Omron CX-Programmer project NuevoProyecto (CX-Programmer 9.80)

# PLC NuevoPLC1: CJ2M CPU34
I/O table (CPU CJ2M-CPU34): rack 0 slot 0 CJ1W-ID211; rack 0 slot 1 CJ1W-ID211; rack 0 slot 2 CJ1W-ID211; rack 0 slot 3 CJ1W-ID211; rack 0 slot 4 CJ1W-OD212; rack 0 slot 5 CJ1W-OD212; rack 0 slot 6 CJ1W-OC211; rack 0 slot 7 CJ1W-CT021; rack 0 slot 11 CJ2M-EIP21

## Global symbols (name address type ; comment)
Alta_vel_Motor_carro_film 6.04 BOOL  ; Alta velocidad del motor de arrastre
Aplicador_desplazado 0.03 BOOL  ; DT. Aplicador desplazado
Aplicador_en_reposo 0.02 BOOL  ; DT. Aplicador en reposo
0.11 BOOL  ; Llave en campo habilita cinta inclinana
0.12 BOOL  ; Run Variador V1 (falla=0)
0.13 BOOL  ; Run variador V2 (falla=0)
0.14 BOOL  ; run variador V3 (falla=0)
0.15 BOOL  ; Señal monitor de tensión (falla=0)
1000.00 BOOL  ; Manual/Automático
1001.00 BOOL  ; Paradas General
108.00 BOOL  ; Entrada de bolsa
10.00 BOOL  ; Ciclo Rodillos - Paso 0 - muevo rodillos
11.00 BOOL  ; Ciclo rodillos - Muevo rodillos hasta centrador
120.00 BOOL  ; Activación de Resto
121.00 BOOL  ; Secuencia resto - Paso 1
122.00 BOOL  ; Secuencia resto - Paso 2
123.00 BOOL  ; Secuencia resto - Paso 3
124.00 BOOL  ; Secuencia resto - Paso 4
125.00 BOOL  ; Secuencia resto  - Paso 5
126.00 BOOL  ; Secuencia resto - Paso 6
128.00 BOOL  ; Se hizo resto
129.00 BOOL  ; Señal fin transferencia enfundadora
12.00 BOOL  ; Ciclo rodillos - Paso 2 -muevo rodillos
135.00 BOOL  ; Deshabilitado
138.00 BOOL  ; Carro pala fin avanse
139.00 BOOL  ; Carro pala - segundo avance
13.00 BOOL  ; Ciclo rodillos - paso 3 - mover Rodillos
144.00 BOOL  ; Primer avance carro pala
145.00 BOOL  ; Segundo avance carro pala
146.00 BOOL  ; Primer avance carro pala
147.00 BOOL  ; segundo avance carro pala
14.00 BOOL  ; Ciclo rodillos - Paso 4 - entrada pallet elevador mover rodillos cuando elevador abajop
150.00 BOOL  ; Sensor
150.01 BOOL  ; Activar bandera
150.05 BOOL  ; Auxiliar Sensor
155.00 BOOL  ; Fin extracto
156.00 BOOL  ; Fin extracto
15.00 BOOL  ; Ciclo rodillos - Paso 5 - Habilita subir pallet, muevo rodillo
16.00 BOOL  ; Ciclo rodillos - paso 6 - muevo rodillos salida pallets
17.00 BOOL  ; Secuencia rodillos - Ultimo paso (necesita puas abajo)
18.00 BOOL  ; Pallet subio en elevador
2000.00 BOOL  ; Alarma por falta de run V1
2000.01 BOOL  ; alarma por falla de run V2
2000.02 BOOL  ; Alarma por falta de run V3
2000.03 BOOL  ; Alarma por falla en alimentación
2000.04 BOOL  ; Alarma por falla de guardamotor D1
2000.05 BOOL  ; Alarma por falla de guardamotor D2
2000.06 BOOL  ; Alarma por falla de gaurdamotor D5
2000.07 BOOL  ; Alarma por falla de guardamotor D7
2000.08 BOOL  ; Alarma por falla variador Elevador
2000.09 BOOL  ; Alarma por falla guardamotor D8L
2000.10 BOOL  ; Alarma por falla guardamotor D9
2000.15 BOOL  ; Falla en motores (termicos)
2001.00 BOOL  ; Flash en HMI
2001.01 BOOL  ; Falla en motores (termicos)
2002.00 BOOL  ; P_emergencia 1 pulsado
2002.01 BOOL  ; P_emergencia 2 pulsado
2002.02 BOOL  ; P_emergencia 3 pulsado
2002.03 BOOL  ; P_emergencia 4 pulsado
2002.04 BOOL  ; Swicht seguridad 1
2002.05 BOOL  ; Swicht seguridad 2
2002.06 BOOL  ; Swicht seguridad 3
2002.07 BOOL  ; Swicht seguridad 4
2002.08 BOOL  ; Swicht seguridad 5
2002.09 BOOL  ; Cortina de seguridad
2002.10 BOOL  ; Contactor alimentación general caido
2002.11 BOOL  ; Discrepancia en entrada de PLC seguridad
2002.12 BOOL  ; Discrepancia en salida de PLC seguridad
2002.13 BOOL  ; Maquina sin seguridad
2002.14 BOOL  ; Barrera inhibida
2002.15 BOOL  ; Pulsador de emregencia pallet vacios pulsada
2003.00 BOOL  ; flash HMI
2004.00 BOOL  ; Pulsador de emergencia escalera
2004.01 BOOL  ; Barrera de seguridad entrada de Pallets
2004.02 BOOL  ; Seguridad de Barrera entrada de Pallets Inhibida
200.00 BOOL  ; Elevador bajar rapido
200.01 BOOL  ; Elevador subir rapido
200.02 BOOL  ; Elevador bajar lento
200.03 BOOL  ; Elevador subir lento
200.05 BOOL  ; Elevador subir rapido
200.06 BOOL  ; Elevador subir rapido
200.07 BOOL  ; Auxiliar freno
2010.00 BOOL  ; Flash en HMI
202.00 BOOL  ; Deformación
2100.00 BOOL  ; Open Gate counter 1
2101.01 BOOL  ; Close gate counter 1
2102.00 BOOL  ; gate open
2102.01 BOOL  ; Gate Close
2102.03 BOOL  ; Reset counter 1
2122 CHANNEL  ; Counter1 (módulo CT021)
250.00 BOOL  ; Habilito  tarea Automatico
250.01 BOOL  ; Habilito tarea Manual
250.02 BOOL  ; Habilito tarea seguridad
29.00 BOOL  ; Auxiliar ciclo elevador - ok para meter pallet
300.00 BOOL  ; Marcha Automático
301.00 BOOL  ; Automático activo
302.00 BOOL  ; M MANUAL
30.00 BOOL  ; Ciclo elevador - paso 0 - bajar lento
31.00 BOOL  ; Ciclo elevador - Paso 1 - Subir rapido
32.00 BOOL  ; Ciclo elevador - Paso 2 - subir rapido
33.00 BOOL  ; Ciclo elevador - subir lento
34.00 BOOL  ; Ciclo elevador - Paso 4 - Bajar lento
35.00 BOOL  ; Ciclo elevador - Paso 5 - Subir lento
36.00 BOOL  ; Ciclo elevador - paso 6 - bajar lento
37.00 BOOL  ; Ciclo elevador - Paso 7 - bajar..lento...rapido
38.00 BOOL  ; Ciclo elevador - Paso 8 - Bajar rapido lento, Fin pallets
39.00 BOOL  ; Cambio de pallets
3.07 BOOL  ; Señal guardamotor D1 (falla=0)
3.08 BOOL  ; Señal guardamotor D2 (falla=0)
3.09 BOOL  ; Señal guardamotor D5 (falla=0)
3.10 BOOL  ; Señal guardamotor D7 (falla=0)
3.11 BOOL  ; Señal guardamotor C8R (falla=0)
3.12 BOOL  ; Señal guardamotor D8L (falla=0)
3.13 BOOL  ; Señal guardamotor D9 (falla=0)
3.15 BOOL  ; FT vacia
400.00 BOOL  ; Función puesta a cero
400.01 BOOL  ; Paso 1 - carro hacia atrás
400.02 BOOL  ; Paso 2 - caro hacia delante libera sensor
400.03 BOOL  ; Paso 3 - Tiempo
400.04 BOOL  ; Paso 4 - Retrocede carro hasta sensor
400.05 BOOL  ; Paso 5 -  reset encoder
400.06 BOOL  ; Paso 6 - Tiempo para poner 0
400.10 BOOL  ; Cero carro OK
401.00 BOOL  ; Baja velocidad carro
401.01 BOOL  ; Velocidad alta de carro
402.00 BOOL  ; Sujeta FIlm (=1 sujetando)
403.00 BOOL  ; Pinzas (=1 cierra)
404.00 BOOL  ; Corte lamina
404.01 BOOL  ; Retorno de cuchilla
405.00 BOOL  ; Auxiliar sensor pallet
405.01 BOOL  ; Auxiliar
408.00 BOOL  ; Film colocado
40.00 BOOL  ; Inicio ciclo pallet
41.00 BOOL  ; Al medio y salir
42.00 BOOL  ; Ya afuera subir
43.00 BOOL  ; Alimentación de pallet
44.00 BOOL  ; Ir abajo y entrar
45.00 BOOL  ; Sensor en medio
46.00 BOOL  ; bolsa colgada
500.00 BOOL  ; Ya salió pallet
501.00 BOOL  ; Terminó secuencia resto
50.00 BOOL  ; Comando cerrar compuerta
51.00 BOOL  ; Comando abrir compuerta
52.00 BOOL  ; Compuerta abierta
54.00 BOOL  ; Bandera para realizar bolsa 4,8,12 y 16
55.00 BOOL  ; Bolsa 4, 8, 12 y 16 en posicion
57.00 BOOL  ; Palet en elevador
58.00 BOOL  ; Activación de barrera
599.14 BOOL  ; P_Off
5.08 BOOL  ; Bandela elevador
600.00 BOOL  ; Activación manual HMI
600.01 BOOL  ; Desactivación Manual HMI
600.02 BOOL  ; Llave Man Aut HMI (1=AUT)
600.04 BOOL  ; Marcha Automático HMI
600.05 BOOL  ; Puesta a cero HMI
600.06 BOOL  ; Resto
600.07 BOOL  ; Cambio de pallets
600.10 BOOL  ; Boton reset HMI
60.00 BOOL  ; Paso 0 - Carro pala Esperando bolsas
610.00 BOOL  ; Manual HMI alimentador
610.01 BOOL  ; Manual HMI Calefactores/ventilalor
610.02 BOOL  ; Manual avance HMI
610.03 BOOL  ; Manual retroceso HMI
610.04 BOOL  ; Manual HMI Prensa
610.05 BOOL  ; Manual pinza HMI
610.06 BOOL  ; Manual corte HMI
610.07 BOOL  ; Manual HMI centrador derecho
610.08 BOOL  ; Manual centrador izquierdo HMI
610.10 BOOL  ; Boton reconocimiento HMI
61.00 BOOL  ; Paso 1 - carro pala avance
62.00 BOOL  ; Paso 2  - carro pala avanza un poco mas (presiona bolsa)
63.00 BOOL  ; paso 3 - Carro pala retroceder
64.00 BOOL  ; Auxiliar sacar banderas de pedido
65.00 BOOL  ; Bandera de realizar avance de carro pala
68.00 BOOL  ; Pulsos de carro pala > Activación de velocidad carro pala
69.00 BOOL  ; Se realizo secuencia avance Bolsa 8 y 16
6.01 BOOL  ; Motor transporte rodillos film
6.14 BOOL  ; Cilindros sujeta Film en elevador
6.15 BOOL  ; Reserva cableada
700.00 BOOL  ; Fin Avance de carro pala (en pulsos)
70.00 BOOL  ; Primera secuencia hecha
72.00 BOOL  ; Seguridad arrastre carro pala
76.00 BOOL  ; Bolsa entrando (filtros con sensores)
77.00 BOOL  ; Pulso para decodificador de movimiento rodillos (bolsas)
800.00 BOOL  ; Auxiliar
82.00 BOOL  ; Pulso bolsa par entrando
86.00 BOOL  ; Rodillos superiores movio OK
87.00 BOOL  ; Bolsas impares
88.00 BOOL  ; Bolsas pares
90.00 BOOL  ; Solicitud de accionamiento de tope de giro
91.00 BOOL  ; Accionar tope de giro (demora encendido)
92.00 BOOL  ; Accionar tope de giro (demora apagado)
93.00 BOOL  ; Solicitud de accionar valvula desplazadora
94.00 BOOL  ; Accionar desplazador
950.00 BOOL  ; M Manual/automático
95.00 BOOL  ; M dosificación
C0014 BOOL  ; C dosificador
D100 CHANNEL  ; Pasos secuencia Maquina Film
D1000 CHANNEL  ; HMI - CANTIDAD DE FILAS POR PALLET
D1002 CHANNEL  ; Filas de pallets
D1003 CHANNEL  ; Activación de velocidad carro pala
D1005 CHANNEL  ; Cantidad pulsos de Avance de carro
D101 CHANNEL  ; Paso anterior
D1012 CHANNEL  ; Pisos en donde se activa la secuencia de carga de pallet
D1014 CHANNEL  ; Pulsos a realizar cinta programada
D200 CHANNEL  ; Programa seleccionado en HMI
D2000 CHANNEL  ; Encoder en milimetros
D2002 CHANNEL  ; Destino en mm de carro
D2004 CHANNEL  ; Largo HMI
D2006 CHANNEL  ; Segundo avance HMI
D2008 CHANNEL  ; Maximo distancia film
D202 CHANNEL  ; Pasos de la secuencia EF
D210 CHANNEL  ; Tiempo desde HMI
D211 CHANNEL  ; Tiempo desde HMI
D212 CHANNEL  ; Tiempo desde HMI
D213 CHANNEL  ; Tiempo desde HMI
D214 CHANNEL  ; Tiempo para seguir arrastre
D300 CHANNEL  ; Decodificador secuencia cargador de pallets
D3100.00 BOOL  ; Comunicacion PLC seg. Inhibir barrera
D3100.01 BOOL  ; Comunicacion PLC seg. Inhibir barrera entrada de Pallets
D3100.02 BOOL  ; Señal para G9SP - Aviso Hay movimmientos
D3100.03 BOOL  ; Señal para G9SP - Espero Inicio de Ciclo de Pallets se habiliat a cargar
D400 CHANNEL  ; Decodificador secuencia rodillos
D406 CHANNEL  ; Tiempo HMI
D410 CHANNEL  ; Decodificador secuencia rodillos salida
D420 CHANNEL  ; Decodificador salida
D500 CHANNEL  ; Bolsa 1
D5000 CHANNEL  ; Contador bolsas
D5002 CHANNEL  ; Bolsas
D5004 CHANNEL  ; Auxiliar
D5006 CHANNEL  ; Rodillos de pallets
D5008 CHANNEL  ; Cantidad de pisos realizados
D501 CHANNEL  ; Bolsa 2
D5010 CHANNEL  ; Cantidad de pisos realizados
D5012 CHANNEL  ; Auxiliar
D5014 CHANNEL  ; Auxiliar
D5016 CHANNEL  ; Auxiliar
D5018 CHANNEL  ; Auxiliar contador 6
D502 CHANNEL  ; Bolsa 3
D5020 CHANNEL  ; Pulsos carro pala
D5022 CHANNEL  ; Auxiliar c7
D5024 CHANNEL  ; Auxiliar c8 (Accionamiento rodillos superiores)
D5026 CHANNEL  ; Pulsos tope de giro
D5028 CHANNEL  ; Auxiliar C11
D503 CHANNEL  ; Bolsa 4
D5030 CHANNEL  ; Demora de accion de desplazador
D5032 CHANNEL  ; Contador cinta programada
D505 CHANNEL  ; Bolsa 6
D507 CHANNEL  ; Bolsa 8
D508 CHANNEL  ; Bolsa 9
D509 CHANNEL  ; Bolsa 10
D510 CHANNEL  ; Bolsa 11
D5100 CHANNEL  ; Contador
D5102 CHANNEL  ; Contador salida
D512 CHANNEL  ; Bolsa 13
D513 CHANNEL  ; Bolsa 14
D514 CHANNEL  ; Bolsa 15
D6000 CHANNEL  ; Pulsos/tiempo para parar rodillos
H0.01 BOOL  ; Pallet Euro=1  Pallet standar=0(HMI)
H0.05 BOOL  ; Enfundadora NO habilitada - HMI
H0.15 BOOL  ; PUENTE 3.15
H10.00 BOOL  ; Habilitacion de Euro Pallet
T0001 BOOL  ; Tiempo, señal habilita salida pallets
T0002 BOOL  ; Elevador abajo
T0003 BOOL  ; Demora de Nivelacion
T0004 BOOL  ; Tiempo de bolsa colgada
T0005 BOOL  ; Tiempo libera fotocelula nivelacion
T0006 BOOL  ; Demora de dosificacion
T0007 BOOL  ; T. compuerta cerrada
T0009 BOOL  ; Tiempo compuerta abierta
T0010 BOOL  ; Tiempo espera pala arriba (filtro)
T0011 BOOL  ; Tiempo carros
T0020 BOOL  ; Tiempo Automático
T0022 BOOL  ; Tiempo centrada
T0030 BOOL  ; Auxiliar freno
T0031 BOOL  ; Auxiliar liberó freno
T0050 BOOL  ; Demora rodillos superior
T0100 BOOL  ; Tiempo apagado ventilador, seguridad calefactores
T0101 BOOL  ; Tiempo centrado longitudinal pallet
T0102 BOOL  ; Tiempo centrado Euro pallet
T0103 BOOL  ; Tiempo espera accionar centrado
T0104 BOOL  ; Tiempo centrado
T0105 BOOL  ; Tiempo centrado
T0106 BOOL  ; Tiempo espera cierre pinzas
T0107 BOOL  ; Espera apertura
T0108 BOOL  ; Tiempo espera corte
T0109 BOOL  ; Tiempo espera avance
T0110 BOOL  ; Tiempo pequeño avance
T0111 BOOL  ; Tiempo espera avance final
T0112 BOOL  ; Tiempo avance sin film
T0113 BOOL  ; Espera retroceso
T0114 BOOL  ; tiempo de calentado film
T0115 BOOL  ; Tiempo calentado film
T0116 BOOL  ; Tiempo falla, pallet trabado
T0120 BOOL  ; Filtro acumulacion de pallets
T0200 BOOL  ; Tiempo auxiliar
T0201 BOOL  ; Tiempo auxiliar
T0202 BOOL  ; Auxiliar
T0203 BOOL  ; Auxiliar
T0204 BOOL  ; Auxiliar
T0205 BOOL  ; Tiempo falla
T0206 BOOL  ; Auxiliar
T0207 BOOL  ; Auxiliar
T0208 BOOL  ; Auxiliar
T0209 BOOL  ; Auxiliar
T0210 BOOL  ; Auxiliar
T0211 BOOL  ; T auxiliar alarma
T0212 BOOL  ; Auxiliar
T0213 BOOL  ; Auxiliar
T0214 BOOL  ; Tiempo para alarma
T0215 BOOL  ; Tiempo para hacer 0
T0216 BOOL  ; T auxiliar alarma
T0217 BOOL  ; Auxiliar
T0218 BOOL  ; Auxiliar
T0219 BOOL  ; Auxiliar
T0220 BOOL  ; Auxiliar
T0221 BOOL  ; Auxiliar
T0222 BOOL  ; Auxiliar
T0223 BOOL  ; Auxiliar
T0224 BOOL  ; Auxiliar no hay pallet
T0225 BOOL  ; Auxiliar
T0226 BOOL  ; Auxiliar
T0227 BOOL  ; Centrador longitudinal
T0228 BOOL  ; Auxiliar tiempo centrador activo
T0229 BOOL  ; Auxiliar
T0230 BOOL  ; auxiliar
T0231 BOOL  ; Auxiliar
T0232 BOOL  ; auxiliar
T0233 BOOL  ; Auxiliar liberacion
T0234 BOOL  ; Auxiliar falla
T0235 BOOL  ; Auxiliar
T0236 BOOL  ; T espera liberación
T0237 BOOL  ; Auxiliar filtro ensor
T0238 BOOL  ; Auxiliar
T0239 BOOL  ; T subir bandela
T0240 BOOL  ; Auxiliar
T0242 BOOL  ; Auxiliar
T0243 BOOL  ; Auxiliar
T0244 BOOL  ; T auxiliar
T1016 BOOL  ; Tiempo de secado de pallets
W12 CHANNEL  ; Salida decodicicador EF
W121.00 BOOL  ; Salida decodificador 3
W121.01 BOOL  ; Salida decodificador 3
W121.02 BOOL  ; Salida decodificador 3
W121.03 BOOL  ; Salida decodificador 3
W121.04 BOOL  ; Salida decodificador 3
W121.05 BOOL  ; Salida decodificador 3
W121.06 BOOL  ; Salida decodificador 3
W121.07 BOOL  ; Salida decodificador 3
W121.08 BOOL  ; Salida decodificador 3
W121.09 BOOL  ; Salida decodificador 3
W121.10 BOOL  ; Salida decodificador 3
W121.11 BOOL  ; Salida decodificador 3
W121.12 BOOL  ; Salida decodificador 3
W121.13 BOOL  ; Salida decodificador 3
W121.14 BOOL  ; Salida decodificador 3
W121.15 BOOL  ; Salida decodificador 3
W150.00 BOOL  ; Paso  0 - Inicio
W150.02 BOOL  ; Paso 2 - Espero OK cinta anterior
W150.04 BOOL  ; Muevo hasta sensor
W150.05 BOOL  ; Paso 5 - Movimiento OK de Cinta
W150.06 BOOL  ; Paso 6 - movimiento OK - Secuencia entrada elevador
W150.08 BOOL  ; Paso 8 - entrar a elevador
W150.10 BOOL  ; Paso 10 - Tiempo
W150.12 BOOL  ; Paso 12 - Pallet dentro de elevador
W150.14 BOOL  ; Paso 14 - movimiento salida
W151.00 BOOL  ; Paso 16 - entrando nuevo pallet
W151.02 BOOL  ; Paso 18 - Pallet ok para elevador
W151.04 BOOL  ; Paso 20 . Salida de pallet
W151.06 BOOL  ; Paso 22 - salida pallets
W151.09 BOOL  ; paso 25 - Alarma pallet trabado
W151.10 BOOL  ; Paso 26 - Alarma de pallet trabado
W200 CHANNEL  ; Canal secuencia maq film
W201 CHANNEL  ; Canal secuencia maq film
W202.00 BOOL  ; Encender cinta rodillos film
W202.01 BOOL  ; Centar pallet derecho Euro
W202.02 BOOL  ; Centar pallet izquierdo Euro
W202.03 BOOL  ; Centar pallet derecho STD
W202.04 BOOL  ; Centar pallets izquierdo STD
W202.05 BOOL  ; Retraer cilindro centrador derecho
W202.06 BOOL  ; Retraer cilindro centrador izquierdo
W202.07 BOOL  ; Val. prensa (mordaza)
W202.08 BOOL  ; Valvula pinzas
W202.09 BOOL  ; Arrastre avance
W202.10 BOOL  ; Motor alimentación film
W202.11 BOOL  ; Corte hacia la izquierda=1 corte hacia la derecha=0
W202.12 BOOL  ; Pequeño avance
W202.13 BOOL  ; Avance sin film (corto)
W202.14 BOOL  ; Arrastre Retroceso
W202.15 BOOL  ; Auxiliar precalentar (paso 2)
W203.00 BOOL  ; Encender rodillos film con rodillos
W203.01 BOOL  ; Habilito secuencia nuevo pallets (habilito finalización de secuencia pallets)
W203.02 BOOL  ; Auxiliar cortar hacia la derecha
W203.03 BOOL  ; Cortador hacia la izquierda
W204.00 BOOL  ; Motor ventilador
W204.01 BOOL  ; Calefactores
W250.01 BOOL  ; Paso 1 - espero
W250.02 BOOL  ; paso 2 -
W250.03 BOOL  ; Paso 3 - Espero reposición enfundadora
W250.04 BOOL  ; paso 4
W250.05 BOOL  ; Paso 5 - Espero OK enfundadora
W300.00 BOOL  ; Paso 0 maquina Film
W300.01 BOOL  ; Paso 1 - Puesta a cero
W300.02 BOOL  ; Paso 2 - Espera de pallets
W300.03 BOOL  ; Paso 3 - movimiento de rodillos
W300.04 BOOL  ; Paso 4 - Centrador de pallets
W300.05 BOOL  ; Paso 5 - Tiempo
W300.06 BOOL  ; Paso 6 - Cierre de pinzas
W300.07 BOOL  ; Paso 7 - Tiempo
W300.08 BOOL  ; Paso 8 - Abre sujeta film
W300.09 BOOL  ; Paso 9 - Primer avance de carro
W300.10 BOOL  ; Paso 10 - Cierre sujetador
W300.11 BOOL  ; Paso 11 - corte de lamina
W300.12 BOOL  ; Paso 12 - Segundo avance
W300.13 BOOL  ; Paso 13 - Abrir pinzas
W300.14 BOOL  ; Paso 14 - termino maq film, cero
W300.15 BOOL  ; Paso 15 - Traslado de pallets
W301.00 BOOL  ; Paso 16
W301.01 BOOL  ; Paso 17
W301.02 BOOL  ; Paso 18
W301.03 BOOL  ; Paso 19
W301.04 BOOL  ; Paso 20
W301.05 BOOL  ; Paso 21
W301.06 BOOL  ; Paso 22
W301.07 BOOL  ; Paso 23
W301.08 BOOL  ; Paso 24
W301.09 BOOL  ; Paso 25
W301.10 BOOL  ; Paso 26
W301.11 BOOL  ; Paso 27
W301.12 BOOL  ; Paso 28
W301.13 BOOL  ; Paso 29
W301.14 BOOL  ; Paso 30
W301.15 BOOL  ; Paso 31
W50.00 BOOL  ; Paso 0 - espero Inicio
W50.01 BOOL  ; Paso 1 -entrar puas
W50.02 BOOL  ; Paso 2 - Bajar puas
W50.03 BOOL  ; Paso 3 - Subir puas medio
W50.04 BOOL  ; Paso 4 - Puas salir
W50.05 BOOL  ; Paso 5 - puas subir
W50.06 BOOL  ; Paso 6 - Pallet listo para sacar - Secuencia cargador
W50.07 BOOL  ; Paso 7 - bajar puas
W50.08 BOOL  ; Paso  8 - Entrar puas
W50.09 BOOL  ; Paso  9 - espero reinicio de ciclo
W50.12 BOOL  ; Pallet trabado
W66.01 BOOL  ; CMD MANUAL - SALIR PRENSA LATERAL
W66.02 BOOL  ; STOP PRENSA LATERAL
W80.00 BOOL  ; Paso  0 - espero inicio
W80.02 BOOL  ; Paso 2 - espero Ok cargador para mover
W80.04 BOOL  ; Paso 4 - muevo cintas
W80.06 BOOL  ; Paso 6 - Ok salio pallet de cargado, Muevo cinta film
W80.08 BOOL  ; Paso 8 - activo centrador
W80.10 BOOL  ; Paso 10 - Espero OK de maq film
W80.12 BOOL  ; Paso 12 - pallet listo para sacar
W80.14 BOOL  ; Paso 14 - Falla, pallet trabajo
W90.00 BOOL  ; Paso  0 - Inicio
W90.02 BOOL  ; Paso 2 - Espero OK cinta anterior
W90.04 BOOL  ; Muevo hasta sensor
W90.06 BOOL  ; Paso 6 - movimiento OK
W90.08 BOOL  ; Paso 8 - entrar a elevador
W90.10 BOOL  ; Paso 10 - Tiempo
W90.12 BOOL  ; Paso 12 - Pallet dentro de elevador
W90.14 BOOL  ; Paso 14 - movimiento salida
Contador_1 Conversion_Encoder
Corte_Activo 0.10 BOOL  ; DT. corte aplicador activado
Corte_en_reposo 0.09 BOOL  ; DT. Cortador en reposo
Estado_entradas_G9SP D3007 CHANNEL  ; Estado entradas PLC seguridad (0=falla bit a bit)
Estado_entradas_G9SP_16_19 D3008 CHANNEL  ; Estado entradas PLC seguridad (0=falla bit a bit)
Estado_salidas_G9SP D3010 CHANNEL  ; Estado salidas PLC seguridad (0=falla bit a bit)
Falla_variador_transportador 3.02 BOOL  ; FC PRENSA LATERAL, POS 1
Fallo_variador_arrastre 3.05 BOOL  ; Falla en variador de arrastre de film
Fi_transferenci_enfundadora 0.08 BOOL  ; Fin de trasferencia de pallets a la enfundadora (señal desde enfundadora)
Hab_FILM H0.00 BOOL  ; Habilitación proceso máquina film
I_G9SP_0 D3002.00 BOOL  ; .
I_G9SP_1 D3002.01 BOOL  ; Entrada PLC Seguridad P_emergencia embolsadora payper
I_G9SP_10 D3002.10 BOOL  ; Entrada PLC Seguridad Cortina seguridad 1
I_G9SP_11 D3002.11 BOOL  ; Entrada PLC Seguridad Cortina seguridad 1
I_G9SP_12 D3002.12 BOOL  ; Entrada PLC Seguridad Contacto modo
I_G9SP_13 D3002.13 BOOL  ; Entrada PLC Seguridad Contacto modo
I_G9SP_14 D3002.14 BOOL  ; Entrada PLC Seguridad Realimentacion relé
I_G9SP_15 D3002.15 BOOL  ; Entrada PLC Seguridad
I_G9SP_16 D3003.00 BOOL  ; Entrada PLC Seguridad
I_G9SP_17 D3003.01 BOOL  ; Entrada PLC Seguridad
I_G9SP_18 D3003.02 BOOL  ; Entrada PLC Seguridad
I_G9SP_19 D3003.03 BOOL  ; Entrada PLC Seguridad
I_G9SP_2 D3002.02 BOOL  ; Entrada PLC Seguridad P_emergencia 2 pallet lleno
I_G9SP_3 D3002.03 BOOL  ; Entrada PLC Seguridad P_emergencia 3 estrichadora
I_G9SP_4 D3002.04 BOOL  ; Entrada PLC Seguridad P_emergencia gabinete comando
I_G9SP_5 D3002.05 BOOL  ; Entrada PLC Seguridad Swicht 1 pallet vacio
I_G9SP_6 D3002.06 BOOL  ; Entrada PLC Seguridad Swicht 2 puerta de elevador
I_G9SP_7 D3002.07 BOOL  ; Entrada PLC Seguridad Swicht 3 pallet lleno
I_G9SP_8 D3002.08 BOOL  ; Entrada PLC Seguridad Swicht 4 puerta tablero neumatico
I_G9SP_9 D3002.09 BOOL  ; Entrada PLC Seguridad Swicht 5 puerta tablero comando
Llave_cinta_inclinada 0.11 BOOL  ; Llave cinta inclinada
M976 W121.00 BOOL  ; Salida decodificador 3
M977 W121.01 BOOL  ; Salida decodificador 3
M978 W121.02 BOOL  ; Salida decodificador 3
M979 W121.03 BOOL  ; Salida decodificador 3
M980 W121.04 BOOL  ; Salida decodificador 3
M981 W121.05 BOOL  ; Salida decodificador 3
M982 W121.06 BOOL  ; Salida decodificador 3
M983 W121.07 BOOL  ; Salida decodificador 3
M984 W121.08 BOOL  ; Salida decodificador 3
M985 W121.09 BOOL  ; Salida decodificador 3
M986 W121.10 BOOL  ; Salida decodificador 3
M987 W121.11 BOOL  ; Salida decodificador 3
M988 W121.12 BOOL  ; Salida decodificador 3
M989 W121.13 BOOL  ; Salida decodificador 3
M990 W121.14 BOOL  ; Salida decodificador 3
M991 W121.15 BOOL  ; Salida decodificador 3
Motor_Rodillos_pallets_vacios 5.13 BOOL  ; Motor transporte de rodillos pallets vacios
Motor_alim_film 6.02 BOOL  ; Motor alimentación de film
Motor_avance 6.05 BOOL  ; Motor de arrastre avance (variador)
Motor_retroceso 6.06 BOOL  ; Motor de arrastre retroceso (variador)
Motor_rodillos_film 6.01 BOOL  ; Motor transporte rodillos film
OLD_M160 160.00 BOOL  ; Programa 1
OLD_M161 160.01 BOOL  ; Programa 2
OLD_M960 W120.00 BOOL  ; Salida decodificador 3
OLD_M961 W120.01 BOOL  ; Salida decodificador 3
OLD_M962 W120.02 BOOL  ; Salida decodificador 3
OLD_M963 W120.03 BOOL  ; Salida decodificador 3
OLD_M964 W120.04 BOOL  ; Salida decodificador 3
OLD_M965 W120.05 BOOL  ; Salida decodificador 3
OLD_M966 W120.06 BOOL  ; Salida decodificador 3
OLD_M967 W120.07 BOOL  ; Salida decodificador 3
OLD_M968 W120.08 BOOL  ; Salida decodificador 3
OLD_M969 W120.09 BOOL  ; Salida decodificador 3
OLD_M970 W120.10 BOOL  ; Salida decodificador 3
OLD_M971 W120.11 BOOL  ; Salida decodificador 3
OLD_M972 W120.12 BOOL  ; Salida decodificador 3
OLD_M973 W120.13 BOOL  ; Salida decodificador 3
OLD_M974 W120.14 BOOL  ; Salida decodificador 3
OLD_M975 W120.15 BOOL  ; Salida decodificador 3
OLD_S0 W0.00 BOOL  ; Salida decodificador
OLD_S1 W0.01 BOOL  ; Salida decodificador - Bolsa 1
OLD_S10 W0.10 BOOL  ; Salida decodificador - Bolsa 10
OLD_S100 W100.00 BOOL  ; Salida decodificador 2
OLD_S101 W100.01 BOOL  ; Salida decodificador 2 Entrada de bolsa
OLD_S102 W100.02 BOOL  ; Salida decodificador 2
OLD_S103 W100.03 BOOL  ; Salida decodificador 2
OLD_S104 W100.04 BOOL  ; Salida decodificador 2
OLD_S105 W100.05 BOOL  ; Salida decodificador 2
OLD_S106 W100.06 BOOL  ; Salida decodificador 2
OLD_S107 W100.07 BOOL  ; Salida decodificador 2
OLD_S108 W100.08 BOOL  ; Salida decodificador 2
OLD_S109 W100.09 BOOL  ; Salida decodificador 2
OLD_S11 W0.11 BOOL  ; Salida decodificador - Bolsa 11
OLD_S110 W100.10 BOOL  ; Salida decodificador 2
OLD_S111 W100.11 BOOL  ; Salida decodificador 2
OLD_S112 W100.12 BOOL  ; Salida decodificador 2
OLD_S113 W100.13 BOOL  ; Salida decodificador 2
OLD_S114 W100.14 BOOL  ; Salida decodificador 2
OLD_S115 W100.15 BOOL  ; Salida decodificador 2
OLD_S116 W101.00 BOOL  ; Salida decodificador 2
OLD_S12 W0.12 BOOL  ; Salida decodificador - Bolsa 12
OLD_S13 W0.13 BOOL  ; Salida decodificador - Bolsa 13
OLD_S14 W0.14 BOOL  ; Salida decodificador - Bolsa 14
OLD_S15 W0.15 BOOL  ; Salida decodificador - Bolsa 15
OLD_S16 W1.00 BOOL  ; Salida decodificador - Bolsa 16
OLD_S2 W0.02 BOOL  ; Salida decodificador - Bolsa 2
OLD_S3 W0.03 BOOL  ; Salida decodificador
OLD_S4 W0.04 BOOL  ; Salida decodificador - Bolsa 4
OLD_S5 W0.05 BOOL  ; Salida decodificador - Bolsa 5
OLD_S6 W0.06 BOOL  ; Salida decodificador - Bolsa 6
OLD_S7 W0.07 BOOL  ; Salida decodificador - Bolsa 7
OLD_S8 W0.08 BOOL  ; Salida decodificador - Bolsa 8
OLD_S9 W0.09 BOOL  ; Salida decodificador - Bolsa 9
OLD_X0 1.00 BOOL  ; Control contaje carro pala
OLD_X16 3.03 BOOL  ; PLC seguridad OK=1
OLD_X27 1.02 BOOL  ; FT acumulación sacos
OLD_X30 1.03 BOOL  ; FT dosificación
OLD_X31 1.04 BOOL  ; FT contaje
OLD_X32 1.05 BOOL  ; FT carros
OLD_X33 1.06 BOOL  ; Pala arriba
OLD_X34 1.07 BOOL  ; Carro pala en reposo
OLD_X35 1.08 BOOL  ; Carro Pala sobre compuerta
OLD_X36 1.09 BOOL  ; Carro pala desplazado
OLD_X37 1.10 BOOL  ; Seguridad arraste carro pala
OLD_X4 1.01 BOOL  ; Seg contrapeso
OLD_X40 1.11 BOOL  ; Compuerta abierta
OLD_X41 1.12 BOOL  ; Compuerta cerrada
OLD_X42 1.13 BOOL  ; Deformación compuerta
OLD_X43 1.14 BOOL  ; Elevador arriba
OLD_X44 1.15 BOOL  ; Elevador cambio velocidad subiendo
OLD_X45 2.00 BOOL  ; Elevador cambio velocidad bajando
OLD_X46 2.01 BOOL  ; elevador abajo
OLD_X47 2.02 BOOL  ; Fotocelula nivelación
OLD_X50 2.03 BOOL  ; Puas dentro
OLD_X51 2.04 BOOL  ; Puas fuera
OLD_X52 2.05 BOOL  ; Puas arriba
OLD_X53 2.06 BOOL  ; Puas centro
OLD_X54 2.07 BOOL  ; Puas abajo
OLD_X55 2.08 BOOL  ; FT. Pallet en espera
OLD_X56 2.09 BOOL  ; FT seguridad entrada elevador
OLD_X57 2.10 BOOL  ; FT pallet en elevador
OLD_X60 2.11 BOOL  ; FT seguridad salida elevador
OLD_X61 2.12 BOOL  ; Acumulación pallets lleno
OLD_X63 2.14 BOOL  ; Presion aire
OLD_X64 2.15 BOOL  ; Valvula desplazadora afuera
OLD_X65 3.00 BOOL  ; Valvula desplazadora adentro
OLD_X66 3.06 BOOL  ; Señal de OK de enfundadora no listo
OLD_Y0 4.00 BOOL  ; Cinta inclinada
OLD_Y1 4.01 BOOL  ; Cinta aplanado superior (Paralaelo inferior)
OLD_Y10 4.08 BOOL  ; Carro pala velocidad 1
OLD_Y11 4.09 BOOL  ; Carro pala velocidad 2
OLD_Y12 4.10 BOOL  ; EV. SALE PRENSA LATERAL
OLD_Y13 4.11 BOOL  ; Desplazador Cinta programada-Alinear. (Válvula)
OLD_Y14 4.12 BOOL  ; Abrir compuerta
OLD_Y15 4.13 BOOL  ; Cerrar compuerta
OLD_Y16 5.00 BOOL  ; Multivelocidad variador (velocidad rápida)
OLD_Y17 5.01 BOOL  ; Freno de elevador
OLD_Y2 4.02 BOOL  ; Cinta Programada
OLD_Y20 4.14 BOOL  ; Elevador subir
OLD_Y21 4.15 BOOL  ; Elevador bajar
OLD_Y22 5.02 BOOL  ; Rodillos palets
OLD_Y23 5.03 BOOL  ; Puas entrar (válvula)
OLD_Y24 5.04 BOOL  ; Puas salir (válvula)
OLD_Y25 5.05 BOOL  ; Puas bajar (válvulas)
OLD_Y26 5.06 BOOL  ; Puas Subir (válvula)
OLD_Y27 5.07 BOOL  ; Barrera (válvula)
OLD_Y3 4.03 BOOL  ; Tope de giro (válvula)
OLD_Y30 6.10 BOOL  ; Centrado pallets (válvula)
OLD_Y31 5.09 BOOL  ; Señal paletizadora en marcha
OLD_Y32 5.10 BOOL  ; Baliza verde
OLD_Y33 5.11 BOOL  ; Baliza Rojo
OLD_Y34 5.12 BOOL  ; EV. ENTRA PRENSA LATERAL
OLD_Y35 6.01 BOOL  ; Salida libre
OLD_Y36 5.14 BOOL  ; Señal para enfundadora - No enfundar
OLD_Y37 5.15 BOOL  ; señal para máquina estrichadora
OLD_Y4 4.04 BOOL  ; Rodillos Superiores
OLD_Y5 4.05 BOOL  ; Pala (válvula)
OLD_Y6 4.06 BOOL  ; Avanzar carro pala
OLD_Y7 4.07 BOOL  ; Retroceder carro pala
O_G9SP_0 D3005.00 BOOL  ; Salida PLC Seguridad Piloto P_emergencia 1
O_G9SP_1 D3005.01 BOOL  ; Salida PLC Seguridad Piloto P_emergencia 2
O_G9SP_2 D3005.02 BOOL  ; Salida PLC Seguridad Piloto P_emergencia 3
O_G9SP_3 D3005.03 BOOL  ; Salida PLC Seguridad Piloto P_emergencia 4
O_G9SP_4 D3005.04 BOOL  ; Salida PLC Seguridad Contactor
O_G9SP_5 D3005.05 BOOL  ; Salida PLC Seguridad
O_G9SP_6 D3005.06 BOOL  ; Salida PLC Seguridad
O_G9SP_7 D3005.07 BOOL  ; Salida PLC Seguridad
P0_film W200.00 BOOL  ; Paso 0 (poner maq en reposo)
P10_film W200.10 BOOL
P11_film W200.11 BOOL
P12_film W200.12 BOOL
P13_film W200.13 BOOL
P14_film W200.14 BOOL
P15_film W200.15 BOOL
P1_film W200.01 BOOL  ; Paso 1 (espera de pallets)
P2_film W200.02 BOOL  ; Centrar pallet transversalmente
P3_film W200.03 BOOL  ; Cierra pinzas y abre mordazas
P4_film W200.04 BOOL  ; Arrastre
P5_film W200.05 BOOL  ; Corte
P6_film W200.06 BOOL  ; pequeño avance
P7_film W200.07 BOOL  ; Retroceso y centrado con calor
P8_film W200.08 BOOL  ; Sacado de pallet a cinta siguiente
P9_film W200.09 BOOL
Pallet_en_cargador 2.13 BOOL  ; Pallet en cargador
Permiso_enfundadora 0.07 BOOL  ; Permiso entrar pallets en enfundadadora
Pres_pallet 0.00 BOOL  ; Presencia de pallet en trasnporte (fotocelda)
Pulsador_abrir_sujetador 0.04 BOOL  ; Llave de habilitación
Pulsador_cerrar_sujetador 0.05 BOOL  ; Pulsador Abrir/Cerrar sujetador de Film
Pulsador_parada_cintas 0.06 BOOL  ; Pulsador parada de cintas
Sensor_control_bobina 0.01 BOOL  ; DT. control bobina aplicador
Termico_arrastre_film 3.04 BOOL  ; Termico de arrastre de film
Termico_trasportador 3.01 BOOL  ; Termico transportador aplicador de film
Val_abrir_pinzas 6.08 BOOL  ; Valvulas abrir pinzas aplicador
Val_abrir_sujetador 6.07 BOOL  ; Valvula abrir sujetador de film
Val_corte 6.09 BOOL  ; Valvula corte lamina aplicador
Valvula_centrador 6.10 BOOL  ; Válvula centrado de pallets vaios
Valvula_centrador_der_no 6.11 BOOL  ; Val. Biestable centrador derecho no accionado
Valvula_cerrar_pinzas 6.13 BOOL  ; Valvula cerrar pinzas aplicador
Valvula_cerrar_sujetador 6.12 BOOL  ; Válvula cerrar sujeta Film aplicador
Velocidad_variador Funcion_baja_velocidad
Ventilador_conveccion 6.03 BOOL  ; Ventilador de aire de convección

## Program General (cyclic task 0)
Local symbols
OLD_M976 BOOL
OLD_X015 BOOL
OLD_X140 BOOL
OLD_X142 BOOL

### Section _Inicio_Salto

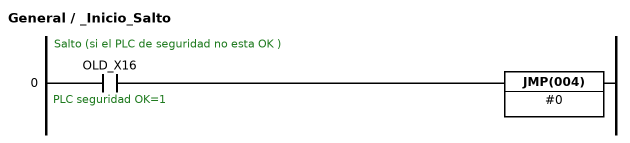
; rung 0: Salto (si el PLC de seguridad no esta OK )
LD OLD_X16  ; PLC seguridad OK=1
JMP(004) #0

### Section Cargador_pallets

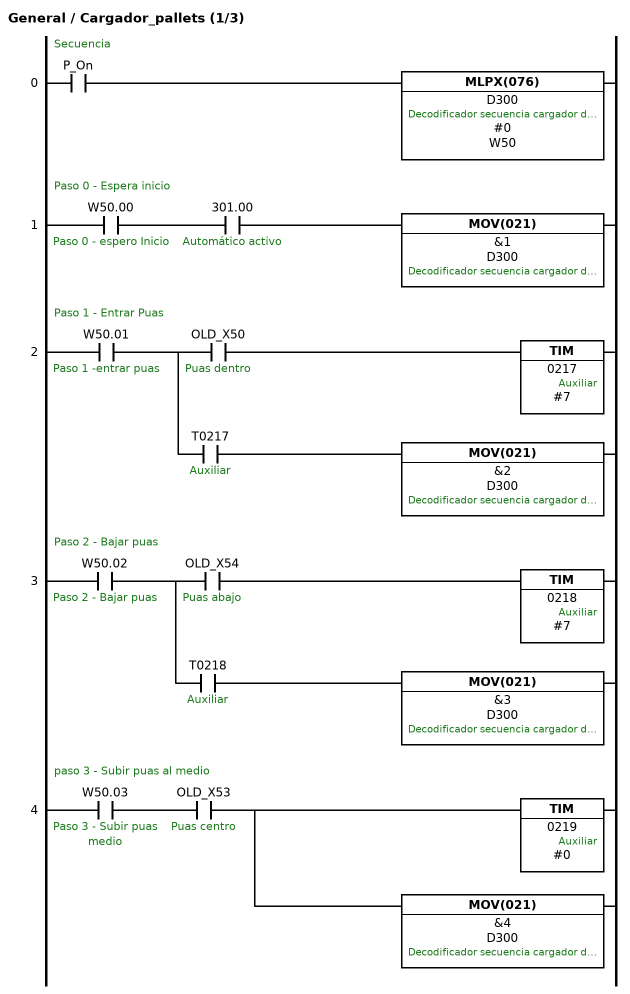
; rung 0: Secuencia
LD P_On
MLPX(076) D300 #0 W50  ; Decodificador secuencia cargador de pallets
; rung 1: Paso 0 - Espera inicio
LD W50.00  ; Paso 0 - espero Inicio
AND 301.00  ; Automático activo
MOV(021) &1 D300  ; Decodificador secuencia cargador de pallets
; rung 2: Paso 1 - Entrar Puas
LD W50.01  ; Paso 1 -entrar puas
OUT TR0
AND OLD_X50  ; Puas dentro
TIM 0217 #7  ; Auxiliar
LD TR0
AND T0217  ; Auxiliar
MOV(021) &2 D300  ; Decodificador secuencia cargador de pallets
; rung 3: Paso 2 - Bajar puas
LD W50.02  ; Paso 2 - Bajar puas
OUT TR0
AND OLD_X54  ; Puas abajo
TIM 0218 #7  ; Auxiliar
LD TR0
AND T0218  ; Auxiliar
MOV(021) &3 D300  ; Decodificador secuencia cargador de pallets
; rung 4: paso 3 - Subir puas al medio
LD W50.03  ; Paso 3 - Subir puas medio
AND OLD_X53  ; Puas centro
TIM 0219 #0  ; Auxiliar
MOV(021) &4 D300  ; Decodificador secuencia cargador de pallets

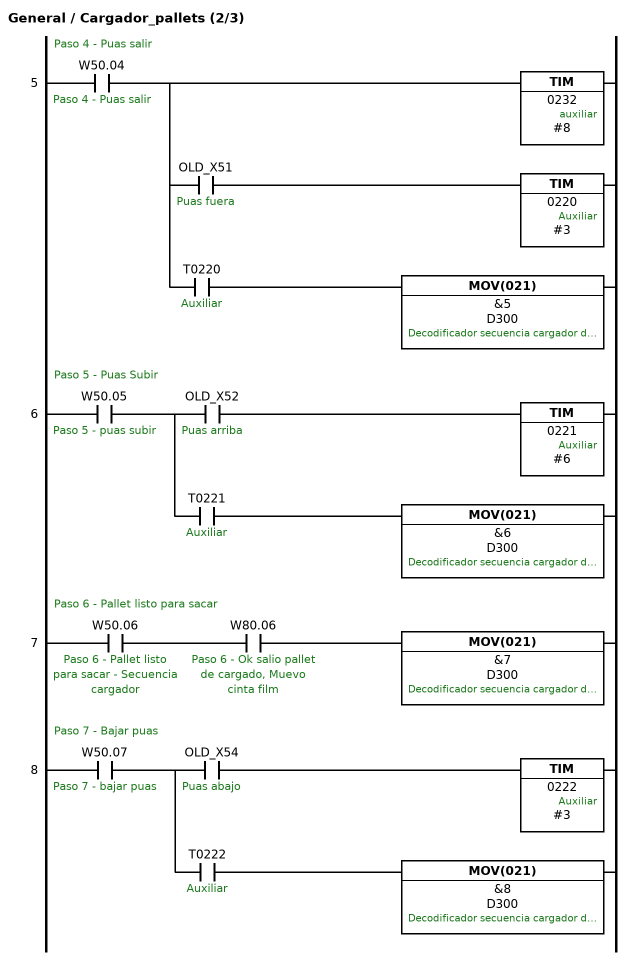
; rung 5: Paso 4 - Puas salir
LD W50.04  ; Paso 4 - Puas salir
OUT TR0
TIM 0232 #8  ; auxiliar
AND OLD_X51  ; Puas fuera
TIM 0220 #3  ; Auxiliar
LD TR0
AND T0220  ; Auxiliar
MOV(021) &5 D300  ; Decodificador secuencia cargador de pallets
; rung 6: Paso 5 - Puas Subir
LD W50.05  ; Paso 5 - puas subir
OUT TR0
AND OLD_X52  ; Puas arriba
TIM 0221 #6  ; Auxiliar
LD TR0
AND T0221  ; Auxiliar
MOV(021) &6 D300  ; Decodificador secuencia cargador de pallets
; rung 7: Paso 6 - Pallet listo para sacar
LD W50.06  ; Paso 6 - Pallet listo para sacar - Secuencia cargador
AND W80.06  ; Paso 6 - Ok salio pallet de cargado, Muevo cinta film
MOV(021) &7 D300  ; Decodificador secuencia cargador de pallets
; rung 8: Paso 7 - Bajar puas
LD W50.07  ; Paso 7 - bajar puas
OUT TR0
AND OLD_X54  ; Puas abajo
TIM 0222 #3  ; Auxiliar
LD TR0
AND T0222  ; Auxiliar
MOV(021) &8 D300  ; Decodificador secuencia cargador de pallets

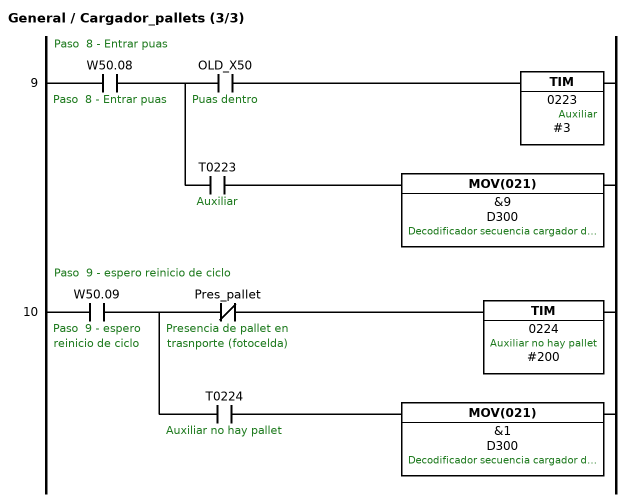
; rung 9: Paso  8 - Entrar puas
LD W50.08  ; Paso  8 - Entrar puas
OUT TR0
AND OLD_X50  ; Puas dentro
TIM 0223 #3  ; Auxiliar
LD TR0
AND T0223  ; Auxiliar
MOV(021) &9 D300  ; Decodificador secuencia cargador de pallets
; rung 10: Paso  9 - espero reinicio de ciclo
LD W50.09  ; Paso  9 - espero reinicio de ciclo
OUT TR0
ANDNOT Pres_pallet  ; Presencia de pallet en trasnporte (fotocelda)
TIM 0224 #200  ; Auxiliar no hay pallet
LD TR0
AND T0224  ; Auxiliar no hay pallet
MOV(021) &1 D300  ; Decodificador secuencia cargador de pallets

### Section Rodillos_centrador

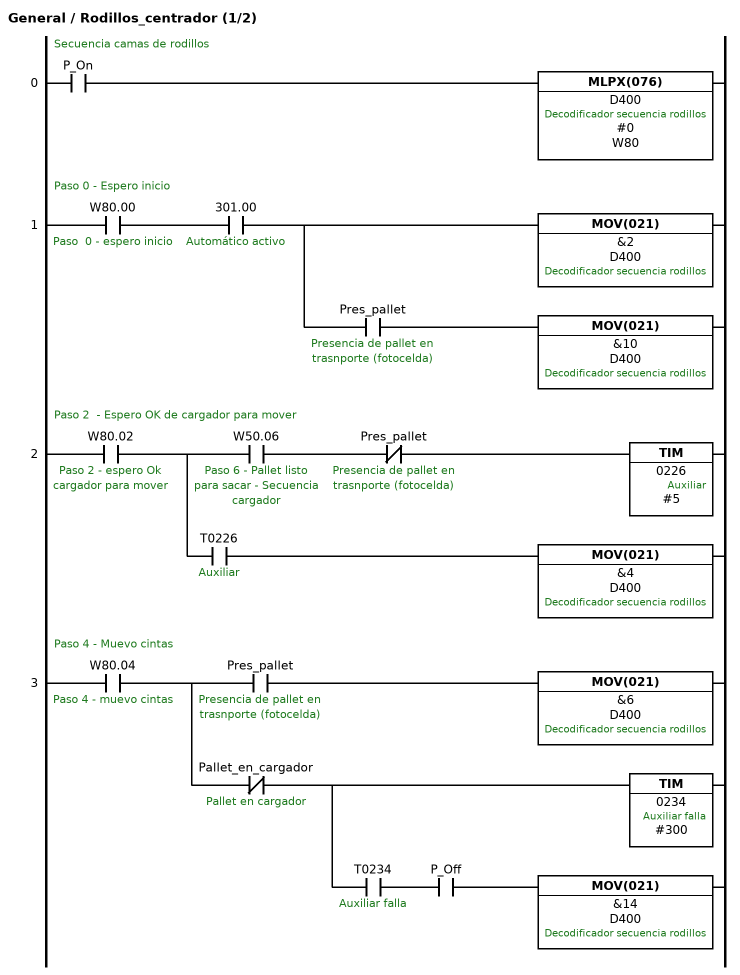
; rung 0: Secuencia camas de rodillos
LD P_On
MLPX(076) D400 #0 W80  ; Decodificador secuencia rodillos
; rung 1: Paso 0 - Espero inicio
LD W80.00  ; Paso  0 - espero inicio
AND 301.00  ; Automático activo
MOV(021) &2 D400  ; Decodificador secuencia rodillos
AND Pres_pallet  ; Presencia de pallet en trasnporte (fotocelda)
MOV(021) &10 D400  ; Decodificador secuencia rodillos
; rung 2: Paso 2  - Espero OK de cargador para mover
LD W80.02  ; Paso 2 - espero Ok cargador para mover
OUT TR0
AND W50.06  ; Paso 6 - Pallet listo para sacar - Secuencia cargador
ANDNOT Pres_pallet  ; Presencia de pallet en trasnporte (fotocelda)
TIM 0226 #5  ; Auxiliar
LD TR0
AND T0226  ; Auxiliar
MOV(021) &4 D400  ; Decodificador secuencia rodillos
; rung 3: Paso 4 - Muevo cintas
LD W80.04  ; Paso 4 - muevo cintas
OUT TR0
AND Pres_pallet  ; Presencia de pallet en trasnporte (fotocelda)
MOV(021) &6 D400  ; Decodificador secuencia rodillos
LD TR0
ANDNOT Pallet_en_cargador  ; Pallet en cargador
TIM 0234 #300  ; Auxiliar falla
AND T0234  ; Auxiliar falla
AND P_Off
MOV(021) &14 D400  ; Decodificador secuencia rodillos

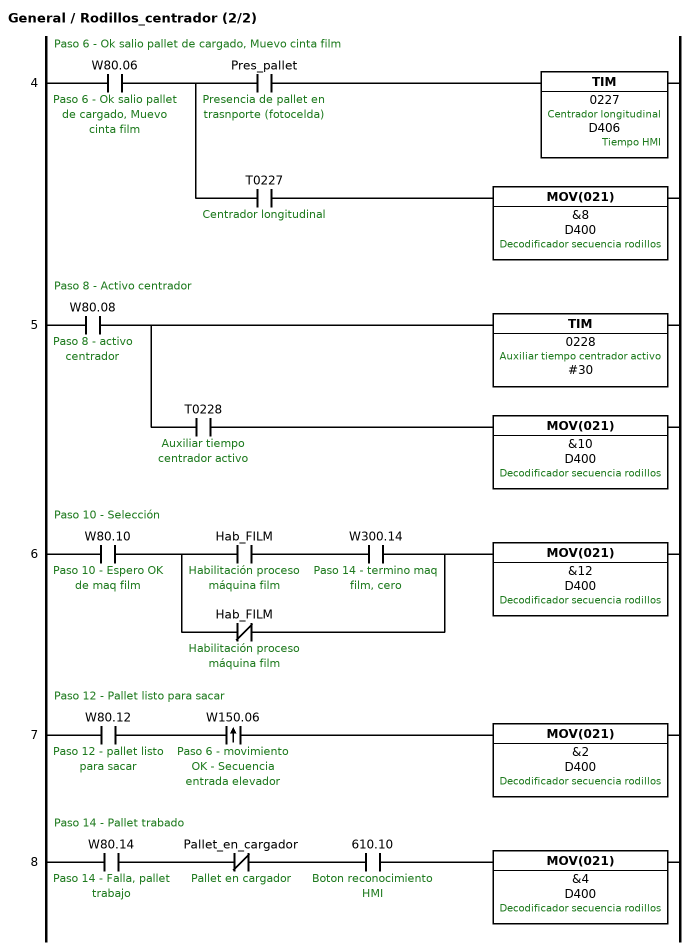
; rung 4: Paso 6 - Ok salio pallet de cargado, Muevo cinta film
LD W80.06  ; Paso 6 - Ok salio pallet de cargado, Muevo cinta film
OUT TR0
AND Pres_pallet  ; Presencia de pallet en trasnporte (fotocelda)
TIM 0227 D406  ; Tiempo HMI, Centrador longitudinal
LD TR0
AND T0227  ; Centrador longitudinal
MOV(021) &8 D400  ; Decodificador secuencia rodillos
; rung 5: Paso 8 - Activo centrador
LD W80.08  ; Paso 8 - activo centrador
TIM 0228 #30  ; Auxiliar tiempo centrador activo
AND T0228  ; Auxiliar tiempo centrador activo
MOV(021) &10 D400  ; Decodificador secuencia rodillos
; rung 6: Paso 10 - Selección
LD W80.10  ; Paso 10 - Espero OK de maq film
LD Hab_FILM  ; Habilitación proceso máquina film
AND W300.14  ; Paso 14 - termino maq film, cero
ORNOT Hab_FILM  ; Habilitación proceso máquina film
ANDLD
MOV(021) &12 D400  ; Decodificador secuencia rodillos
; rung 7: Paso 12 - Pallet listo para sacar
LD W80.12  ; Paso 12 - pallet listo para sacar
@AND W150.06  ; Paso 6 - movimiento OK - Secuencia entrada elevador
MOV(021) &2 D400  ; Decodificador secuencia rodillos
; rung 8: Paso 14 - Pallet trabado
LD W80.14  ; Paso 14 - Falla, pallet trabajo
ANDNOT Pallet_en_cargador  ; Pallet en cargador
AND 610.10  ; Boton reconocimiento HMI
MOV(021) &4 D400  ; Decodificador secuencia rodillos

### Section Rodillos_entrada_elevador

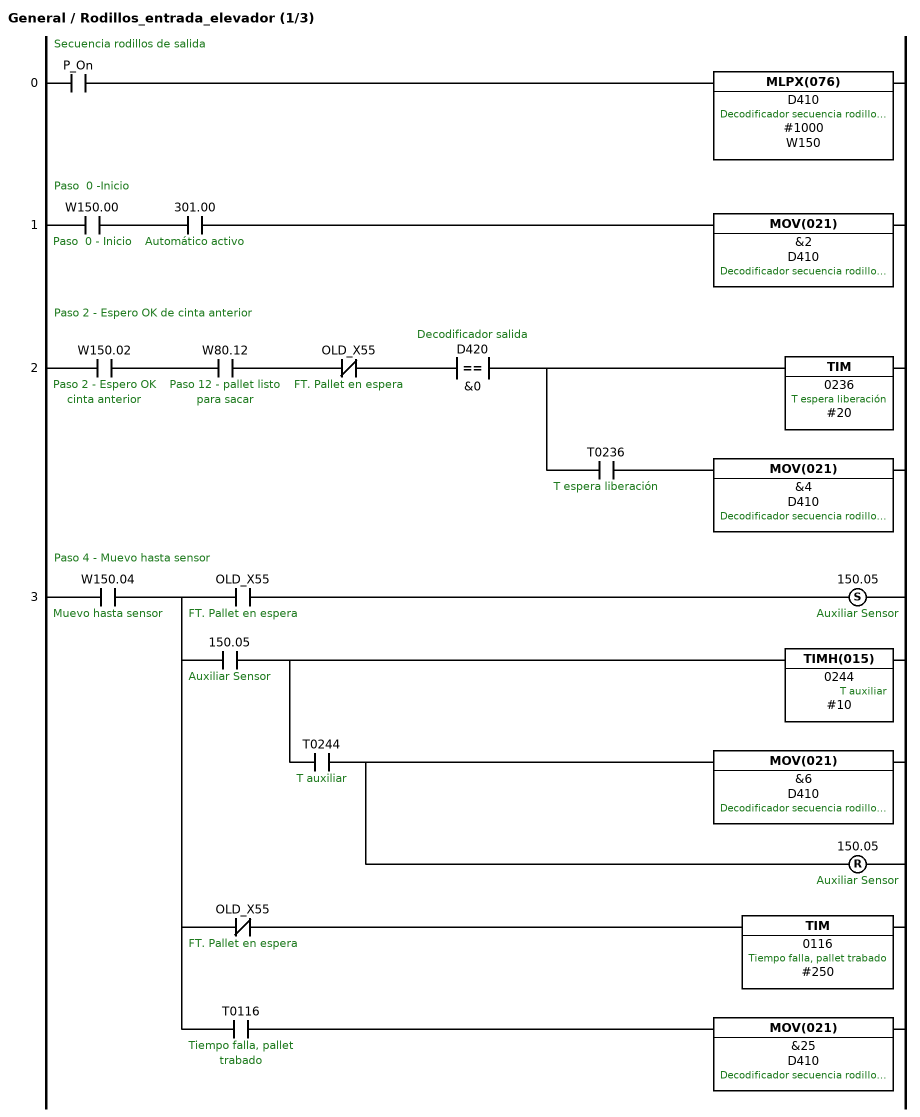
; rung 0: Secuencia rodillos de salida
LD P_On
MLPX(076) D410 #1000 W150  ; Decodificador secuencia rodillos salida
; rung 1: Paso  0 -Inicio
LD W150.00  ; Paso  0 - Inicio
AND 301.00  ; Automático activo
MOV(021) &2 D410  ; Decodificador secuencia rodillos salida
; rung 2: Paso 2 - Espero OK de cinta anterior
LD W150.02  ; Paso 2 - Espero OK cinta anterior
AND W80.12  ; Paso 12 - pallet listo para sacar
ANDNOT OLD_X55  ; FT. Pallet en espera
AND=(300) D420 &0  ; Decodificador salida
TIM 0236 #20  ; T espera liberación
AND T0236  ; T espera liberación
MOV(021) &4 D410  ; Decodificador secuencia rodillos salida
; rung 3: Paso 4 - Muevo hasta sensor
LD W150.04  ; Muevo hasta sensor
OUT TR0
AND OLD_X55  ; FT. Pallet en espera
SET 150.05  ; Auxiliar Sensor
LD TR0
AND 150.05  ; Auxiliar Sensor
TIMH(015) 0244 #10  ; T auxiliar
AND T0244  ; T auxiliar
MOV(021) &6 D410  ; Decodificador secuencia rodillos salida
RSET 150.05  ; Auxiliar Sensor
LD TR0
ANDNOT OLD_X55  ; FT. Pallet en espera
TIM 0116 #250  ; Tiempo falla, pallet trabado
LD TR0
AND T0116  ; Tiempo falla, pallet trabado
MOV(021) &25 D410  ; Decodificador secuencia rodillos salida

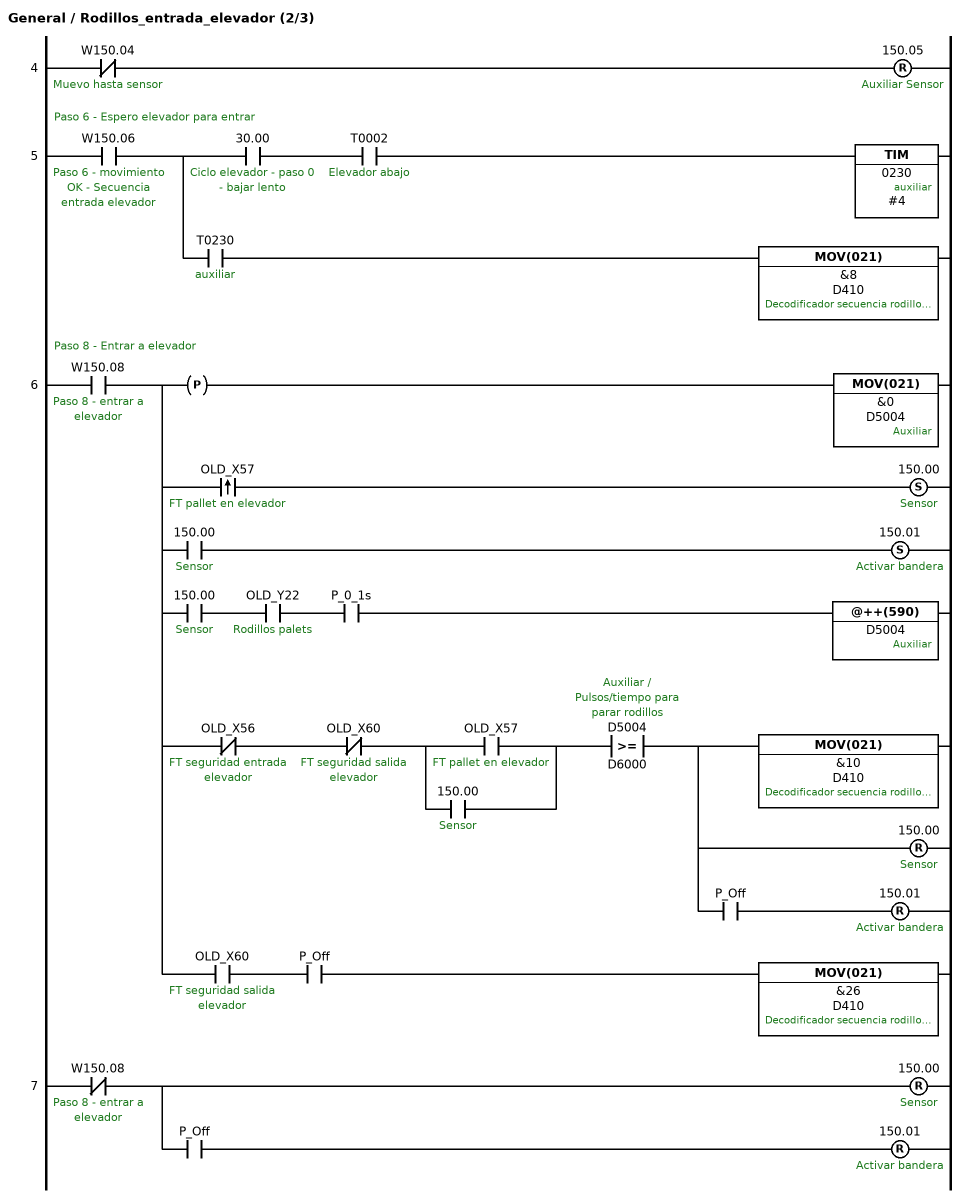
; rung 4
LDNOT W150.04  ; Muevo hasta sensor
RSET 150.05  ; Auxiliar Sensor
; rung 5: Paso 6 - Espero elevador para entrar
LD W150.06  ; Paso 6 - movimiento OK - Secuencia entrada elevador
OUT TR0
AND 30.00  ; Ciclo elevador - paso 0 - bajar lento
AND T0002  ; Elevador abajo
TIM 0230 #4  ; auxiliar
LD TR0
AND T0230  ; auxiliar
MOV(021) &8 D410  ; Decodificador secuencia rodillos salida
; rung 6: Paso 8 - Entrar a elevador
LD W150.08  ; Paso 8 - entrar a elevador
OUT TR0
UP(521)
MOV(021) &0 D5004  ; Auxiliar
LD TR0
@AND OLD_X57  ; FT pallet en elevador
SET 150.00  ; Sensor
LD TR0
AND 150.00  ; Sensor
SET 150.01  ; Activar bandera
LD TR0
AND 150.00  ; Sensor
AND OLD_Y22  ; Rodillos palets
AND P_0_1s
@++(590) D5004  ; Auxiliar
LD TR0
ANDNOT OLD_X56  ; FT seguridad entrada elevador
ANDNOT OLD_X60  ; FT seguridad salida elevador
LD OLD_X57  ; FT pallet en elevador
OR 150.00  ; Sensor
ANDLD
AND>=(325) D5004 D6000  ; Auxiliar, Pulsos/tiempo para parar rodillos
MOV(021) &10 D410  ; Decodificador secuencia rodillos salida
RSET 150.00  ; Sensor
AND P_Off
RSET 150.01  ; Activar bandera
LD TR0
AND OLD_X60  ; FT seguridad salida elevador
AND P_Off
MOV(021) &26 D410  ; Decodificador secuencia rodillos salida
; rung 7
LDNOT W150.08  ; Paso 8 - entrar a elevador
RSET 150.00  ; Sensor
AND P_Off
RSET 150.01  ; Activar bandera

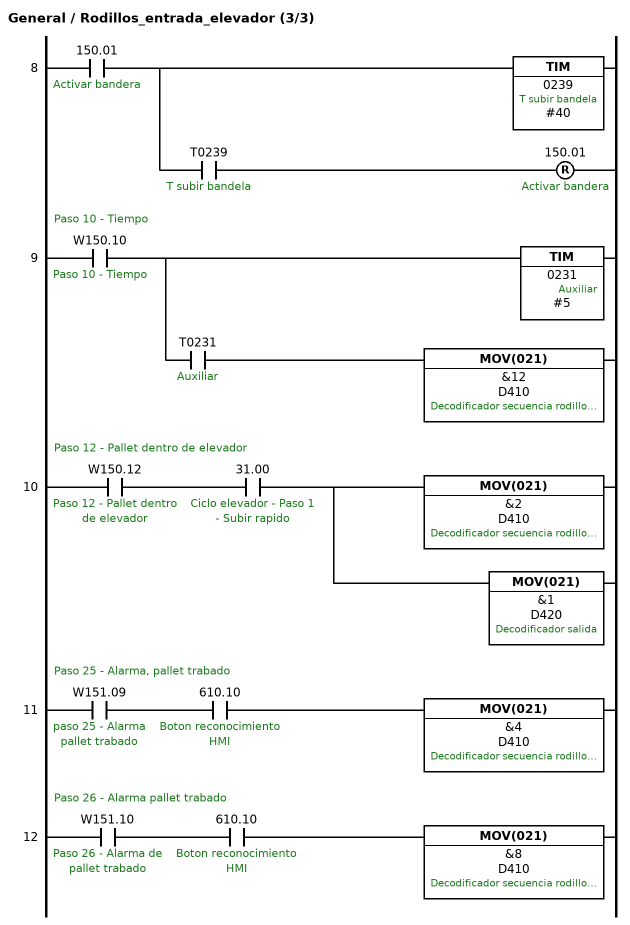
; rung 8
LD 150.01  ; Activar bandera
TIM 0239 #40  ; T subir bandela
AND T0239  ; T subir bandela
RSET 150.01  ; Activar bandera
; rung 9: Paso 10 - Tiempo
LD W150.10  ; Paso 10 - Tiempo
TIM 0231 #5  ; Auxiliar
AND T0231  ; Auxiliar
MOV(021) &12 D410  ; Decodificador secuencia rodillos salida
; rung 10: Paso 12 - Pallet dentro de elevador
LD W150.12  ; Paso 12 - Pallet dentro de elevador
AND 31.00  ; Ciclo elevador - Paso 1 - Subir rapido
MOV(021) &2 D410  ; Decodificador secuencia rodillos salida
MOV(021) &1 D420  ; Decodificador salida
; rung 11: Paso 25 - Alarma, pallet trabado
LD W151.09  ; paso 25 - Alarma pallet trabado
AND 610.10  ; Boton reconocimiento HMI
MOV(021) &4 D410  ; Decodificador secuencia rodillos salida
; rung 12: Paso 26 - Alarma pallet trabado
LD W151.10  ; Paso 26 - Alarma de pallet trabado
AND 610.10  ; Boton reconocimiento HMI
MOV(021) &8 D410  ; Decodificador secuencia rodillos salida

### Section Rodillo_salida

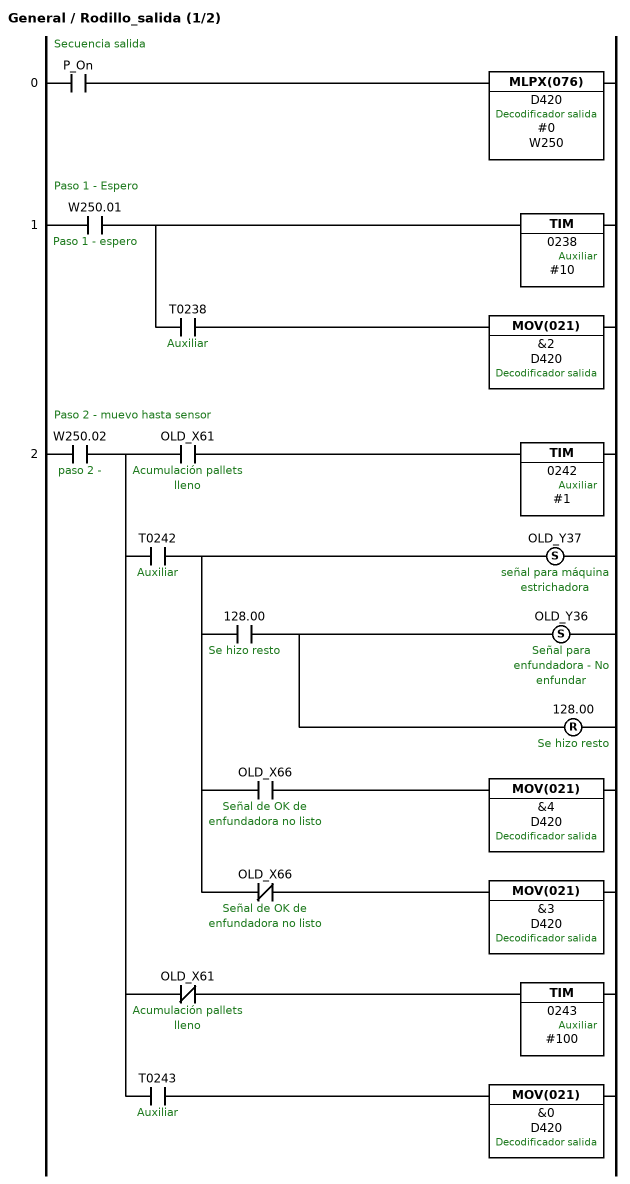
; rung 0: Secuencia salida
LD P_On
MLPX(076) D420 #0 W250  ; Decodificador salida
; rung 1: Paso 1 - Espero
LD W250.01  ; Paso 1 - espero
TIM 0238 #10  ; Auxiliar
AND T0238  ; Auxiliar
MOV(021) &2 D420  ; Decodificador salida
; rung 2: Paso 2 - muevo hasta sensor
LD W250.02  ; paso 2 -
OUT TR0
AND OLD_X61  ; Acumulación pallets lleno
TIM 0242 #1  ; Auxiliar
LD TR0
AND T0242  ; Auxiliar
OUT TR1
SET OLD_Y37  ; señal para máquina estrichadora
AND 128.00  ; Se hizo resto
SET OLD_Y36  ; Señal para enfundadora - No enfundar
RSET 128.00  ; Se hizo resto
LD TR1
AND OLD_X66  ; Señal de OK de enfundadora no listo
MOV(021) &4 D420  ; Decodificador salida
LD TR1
ANDNOT OLD_X66  ; Señal de OK de enfundadora no listo
MOV(021) &3 D420  ; Decodificador salida
LD TR0
ANDNOT OLD_X61  ; Acumulación pallets lleno
TIM 0243 #100  ; Auxiliar
LD TR0
AND T0243  ; Auxiliar
MOV(021) &0 D420  ; Decodificador salida

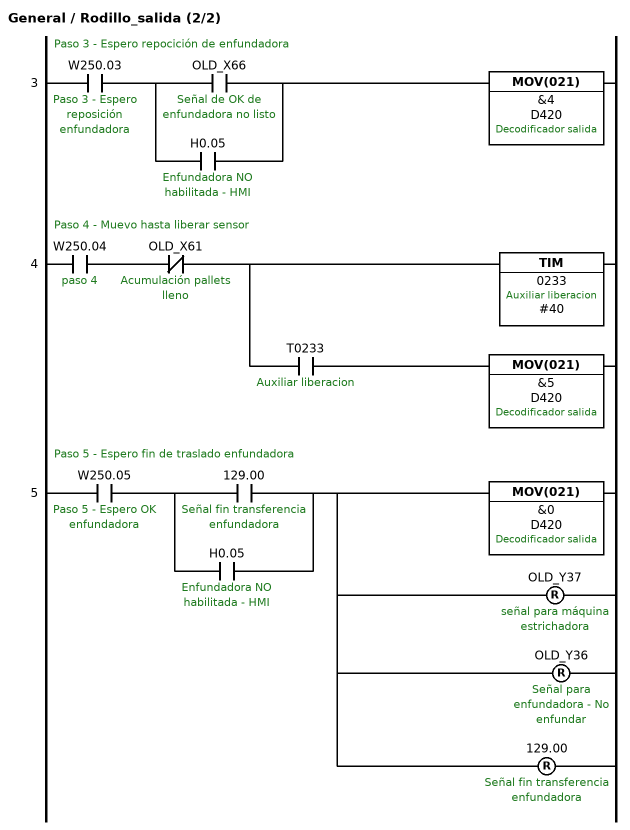
; rung 3: Paso 3 - Espero repocición de enfundadora
LD W250.03  ; Paso 3 - Espero reposición enfundadora
LD OLD_X66  ; Señal de OK de enfundadora no listo
OR H0.05  ; Enfundadora NO habilitada - HMI
ANDLD
MOV(021) &4 D420  ; Decodificador salida
; rung 4: Paso 4 - Muevo hasta liberar sensor
LD W250.04  ; paso 4
ANDNOT OLD_X61  ; Acumulación pallets lleno
TIM 0233 #40  ; Auxiliar liberacion
AND T0233  ; Auxiliar liberacion
MOV(021) &5 D420  ; Decodificador salida
; rung 5: Paso 5 - Espero fin de traslado enfundadora
LD W250.05  ; Paso 5 - Espero OK enfundadora
LD 129.00  ; Señal fin transferencia enfundadora
OR H0.05  ; Enfundadora NO habilitada - HMI
ANDLD
MOV(021) &0 D420  ; Decodificador salida
RSET OLD_Y37  ; señal para máquina estrichadora
RSET OLD_Y36  ; Señal para enfundadora - No enfundar
RSET 129.00  ; Señal fin transferencia enfundadora

### Section Elevador

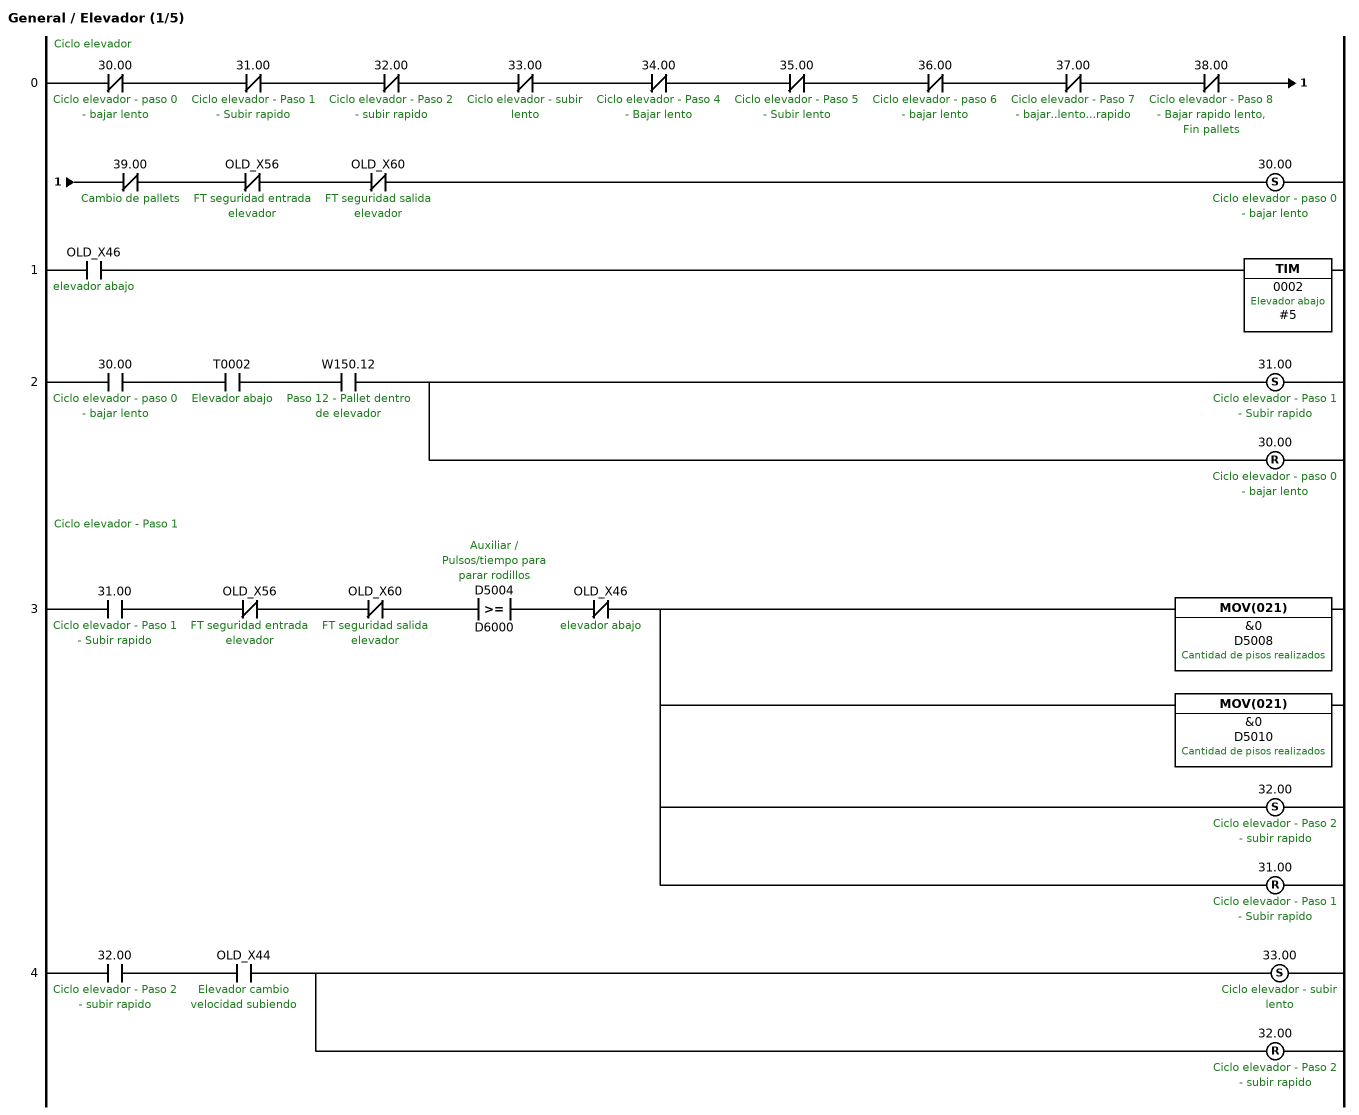
; rung 0: Ciclo elevador
LDNOT 30.00  ; Ciclo elevador - paso 0 - bajar lento
ANDNOT 31.00  ; Ciclo elevador - Paso 1 - Subir rapido
ANDNOT 32.00  ; Ciclo elevador - Paso 2 - subir rapido
ANDNOT 33.00  ; Ciclo elevador - subir lento
ANDNOT 34.00  ; Ciclo elevador - Paso 4 - Bajar lento
ANDNOT 35.00  ; Ciclo elevador - Paso 5 - Subir lento
ANDNOT 36.00  ; Ciclo elevador - paso 6 - bajar lento
ANDNOT 37.00  ; Ciclo elevador - Paso 7 - bajar..lento...rapido
ANDNOT 38.00  ; Ciclo elevador - Paso 8 - Bajar rapido lento, Fin pallets
ANDNOT 39.00  ; Cambio de pallets
ANDNOT OLD_X56  ; FT seguridad entrada elevador
ANDNOT OLD_X60  ; FT seguridad salida elevador
SET 30.00  ; Ciclo elevador - paso 0 - bajar lento
; rung 1
LD OLD_X46  ; elevador abajo
TIM 0002 #5  ; Elevador abajo
; rung 2
LD 30.00  ; Ciclo elevador - paso 0 - bajar lento
AND T0002  ; Elevador abajo
AND W150.12  ; Paso 12 - Pallet dentro de elevador
SET 31.00  ; Ciclo elevador - Paso 1 - Subir rapido
RSET 30.00  ; Ciclo elevador - paso 0 - bajar lento
; rung 3: Ciclo elevador - Paso 1
LD 31.00  ; Ciclo elevador - Paso 1 - Subir rapido
ANDNOT OLD_X56  ; FT seguridad entrada elevador
ANDNOT OLD_X60  ; FT seguridad salida elevador
AND>=(325) D5004 D6000  ; Auxiliar, Pulsos/tiempo para parar rodillos
ANDNOT OLD_X46  ; elevador abajo
MOV(021) &0 D5008  ; Cantidad de pisos realizados
MOV(021) &0 D5010  ; Cantidad de pisos realizados
SET 32.00  ; Ciclo elevador - Paso 2 - subir rapido
RSET 31.00  ; Ciclo elevador - Paso 1 - Subir rapido
; rung 4
LD 32.00  ; Ciclo elevador - Paso 2 - subir rapido
AND OLD_X44  ; Elevador cambio velocidad subiendo
SET 33.00  ; Ciclo elevador - subir lento
RSET 32.00  ; Ciclo elevador - Paso 2 - subir rapido

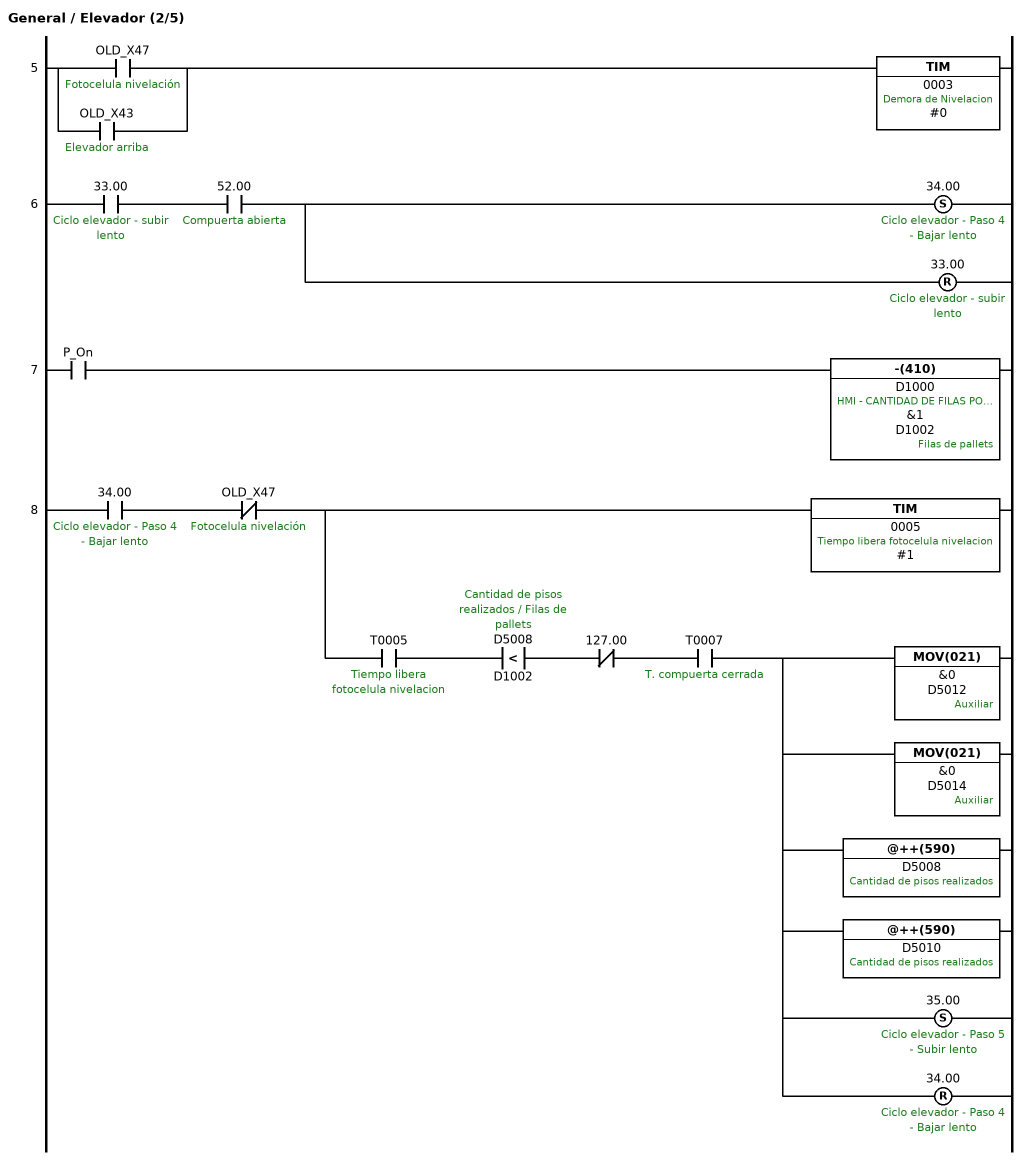
; rung 5
LD OLD_X47  ; Fotocelula nivelación
OR OLD_X43  ; Elevador arriba
TIM 0003 #0  ; Demora de Nivelacion
; rung 6
LD 33.00  ; Ciclo elevador - subir lento
AND 52.00  ; Compuerta abierta
SET 34.00  ; Ciclo elevador - Paso 4 - Bajar lento
RSET 33.00  ; Ciclo elevador - subir lento
; rung 7
LD P_On
-(410) D1000 &1 D1002  ; HMI - CANTIDAD DE FILAS POR PALLET, Filas de pallets
; rung 8
LD 34.00  ; Ciclo elevador - Paso 4 - Bajar lento
ANDNOT OLD_X47  ; Fotocelula nivelación
TIM 0005 #1  ; Tiempo libera fotocelula nivelacion
AND T0005  ; Tiempo libera fotocelula nivelacion
AND<(310) D5008 D1002  ; Cantidad de pisos realizados, Filas de pallets
ANDNOT 127.00
AND T0007  ; T. compuerta cerrada
MOV(021) &0 D5012  ; Auxiliar
MOV(021) &0 D5014  ; Auxiliar
@++(590) D5008  ; Cantidad de pisos realizados
@++(590) D5010  ; Cantidad de pisos realizados
SET 35.00  ; Ciclo elevador - Paso 5 - Subir lento
RSET 34.00  ; Ciclo elevador - Paso 4 - Bajar lento

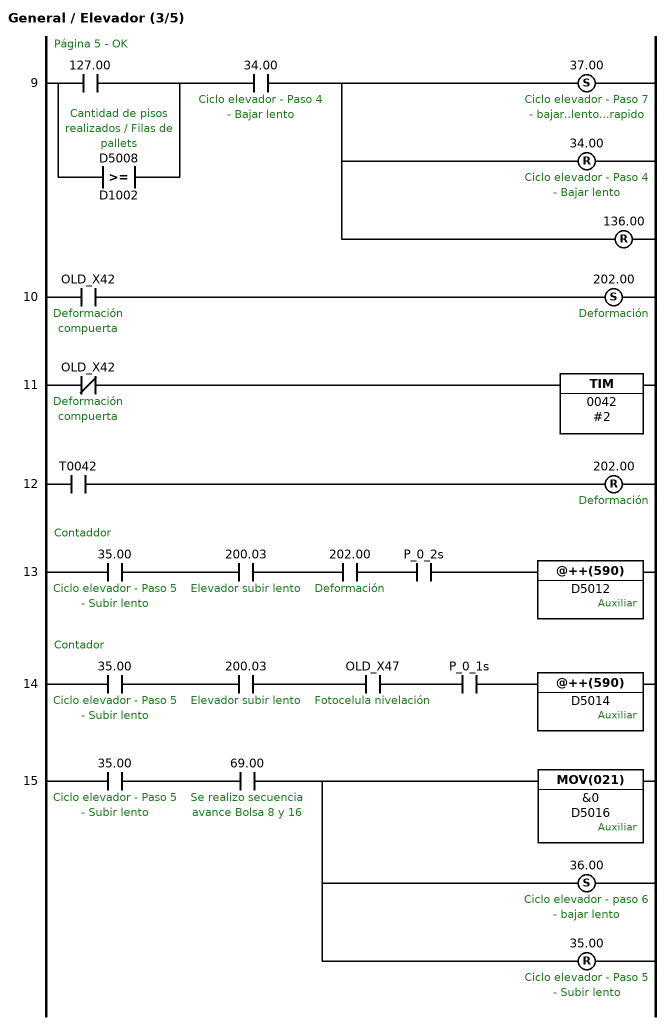
; rung 9: Página 5 - OK
LD 127.00
OR>=(325) D5008 D1002  ; Cantidad de pisos realizados, Filas de pallets
AND 34.00  ; Ciclo elevador - Paso 4 - Bajar lento
SET 37.00  ; Ciclo elevador - Paso 7 - bajar..lento...rapido
RSET 34.00  ; Ciclo elevador - Paso 4 - Bajar lento
RSET 136.00
; rung 10
LD OLD_X42  ; Deformación compuerta
SET 202.00  ; Deformación
; rung 11
LDNOT OLD_X42  ; Deformación compuerta
TIM 0042 #2
; rung 12
LD T0042
RSET 202.00  ; Deformación
; rung 13: Contaddor
LD 35.00  ; Ciclo elevador - Paso 5 - Subir lento
AND 200.03  ; Elevador subir lento
AND 202.00  ; Deformación
AND P_0_2s
@++(590) D5012  ; Auxiliar
; rung 14: Contador
LD 35.00  ; Ciclo elevador - Paso 5 - Subir lento
AND 200.03  ; Elevador subir lento
AND OLD_X47  ; Fotocelula nivelación
AND P_0_1s
@++(590) D5014  ; Auxiliar
; rung 15
LD 35.00  ; Ciclo elevador - Paso 5 - Subir lento
AND 69.00  ; Se realizo secuencia avance Bolsa 8 y 16
MOV(021) &0 D5016  ; Auxiliar
SET 36.00  ; Ciclo elevador - paso 6 - bajar lento
RSET 35.00  ; Ciclo elevador - Paso 5 - Subir lento

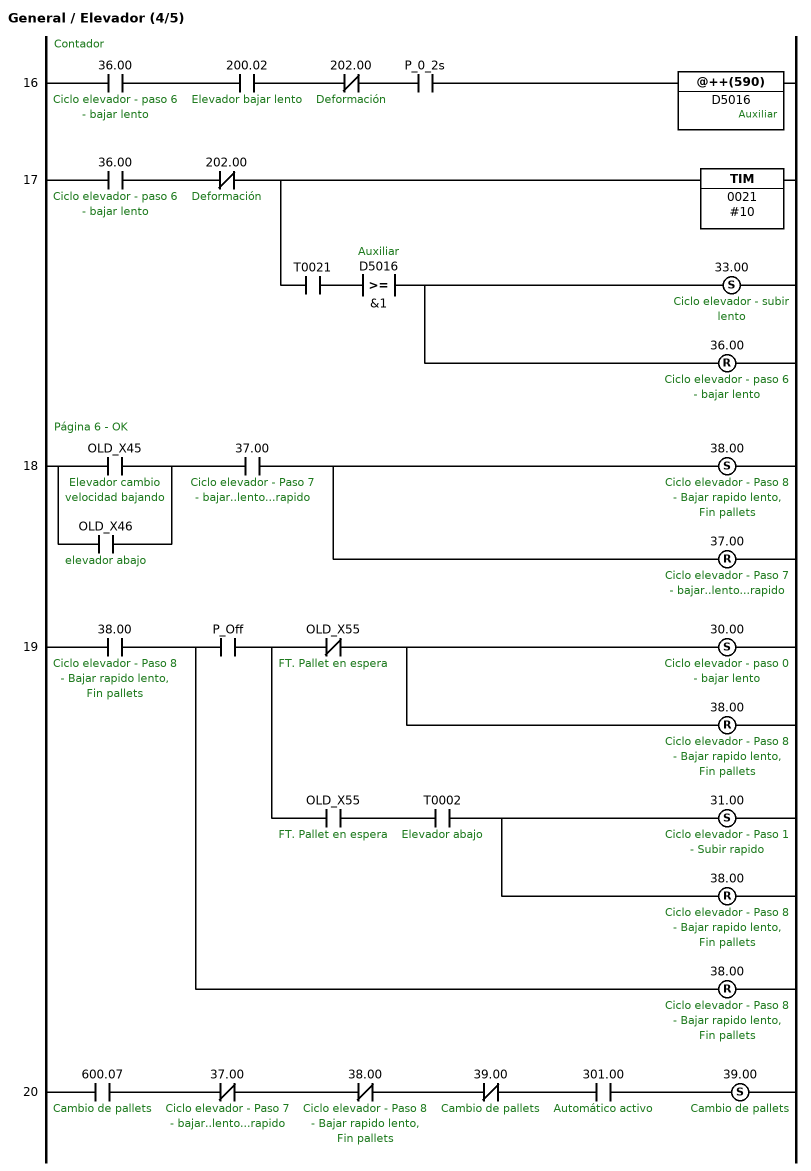
; rung 16: Contador
LD 36.00  ; Ciclo elevador - paso 6 - bajar lento
AND 200.02  ; Elevador bajar lento
ANDNOT 202.00  ; Deformación
AND P_0_2s
@++(590) D5016  ; Auxiliar
; rung 17
LD 36.00  ; Ciclo elevador - paso 6 - bajar lento
ANDNOT 202.00  ; Deformación
TIM 0021 #10
AND T0021
AND>=(325) D5016 &1  ; Auxiliar
SET 33.00  ; Ciclo elevador - subir lento
RSET 36.00  ; Ciclo elevador - paso 6 - bajar lento
; rung 18: Página 6 - OK
LD OLD_X45  ; Elevador cambio velocidad bajando
OR OLD_X46  ; elevador abajo
AND 37.00  ; Ciclo elevador - Paso 7 - bajar..lento...rapido
SET 38.00  ; Ciclo elevador - Paso 8 - Bajar rapido lento, Fin pallets
RSET 37.00  ; Ciclo elevador - Paso 7 - bajar..lento...rapido
; rung 19
LD 38.00  ; Ciclo elevador - Paso 8 - Bajar rapido lento, Fin pallets
OUT TR0
AND P_Off
OUT TR1
ANDNOT OLD_X55  ; FT. Pallet en espera
SET 30.00  ; Ciclo elevador - paso 0 - bajar lento
RSET 38.00  ; Ciclo elevador - Paso 8 - Bajar rapido lento, Fin pallets
LD TR1
AND OLD_X55  ; FT. Pallet en espera
AND T0002  ; Elevador abajo
SET 31.00  ; Ciclo elevador - Paso 1 - Subir rapido
RSET 38.00  ; Ciclo elevador - Paso 8 - Bajar rapido lento, Fin pallets
LD TR0
RSET 38.00  ; Ciclo elevador - Paso 8 - Bajar rapido lento, Fin pallets
; rung 20
LD 600.07  ; Cambio de pallets
ANDNOT 37.00  ; Ciclo elevador - Paso 7 - bajar..lento...rapido
ANDNOT 38.00  ; Ciclo elevador - Paso 8 - Bajar rapido lento, Fin pallets
ANDNOT 39.00  ; Cambio de pallets
AND 301.00  ; Automático activo
SET 39.00  ; Cambio de pallets

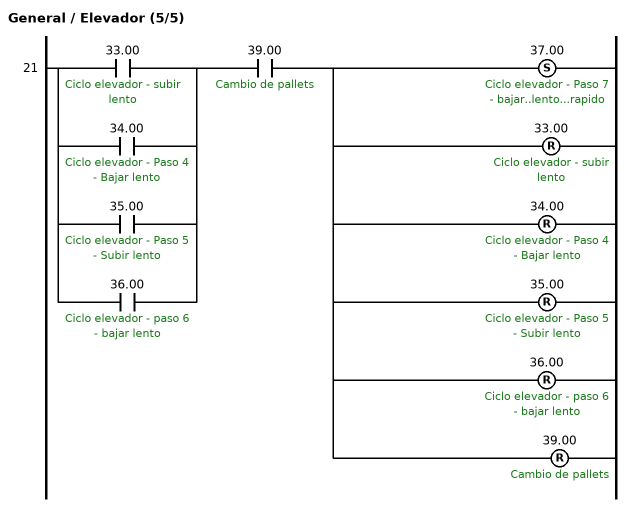
; rung 21
LD 33.00  ; Ciclo elevador - subir lento
OR 34.00  ; Ciclo elevador - Paso 4 - Bajar lento
OR 35.00  ; Ciclo elevador - Paso 5 - Subir lento
OR 36.00  ; Ciclo elevador - paso 6 - bajar lento
AND 39.00  ; Cambio de pallets
SET 37.00  ; Ciclo elevador - Paso 7 - bajar..lento...rapido
RSET 33.00  ; Ciclo elevador - subir lento
RSET 34.00  ; Ciclo elevador - Paso 4 - Bajar lento
RSET 35.00  ; Ciclo elevador - Paso 5 - Subir lento
RSET 36.00  ; Ciclo elevador - paso 6 - bajar lento
RSET 39.00  ; Cambio de pallets

### Section Maquina_de_Film

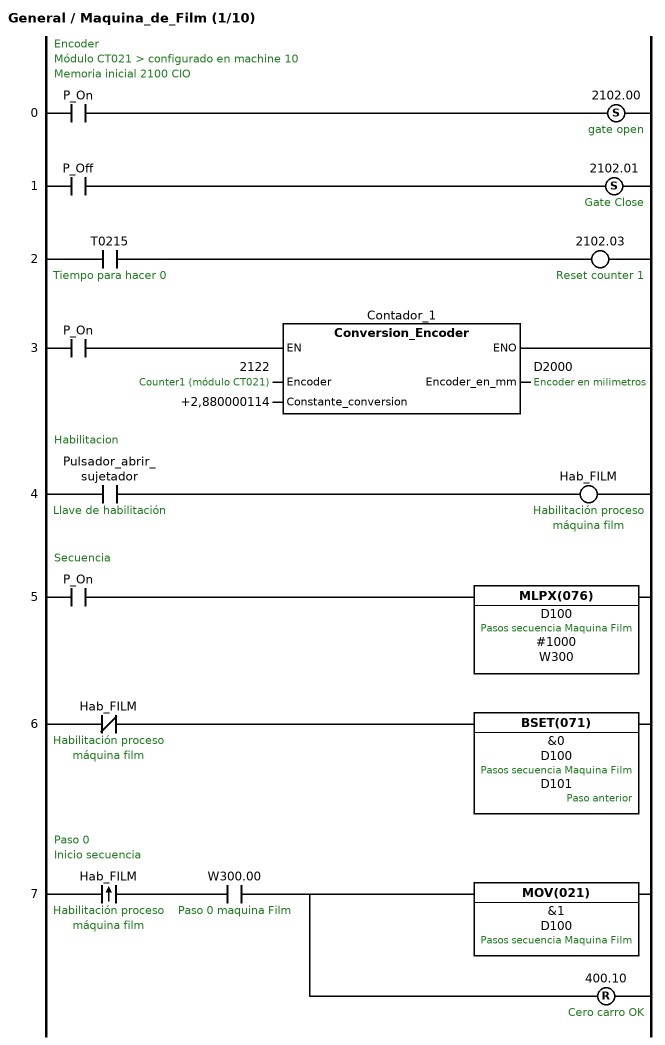
; rung 0: Encoder / Módulo CT021 > configurado en machine 10 / Memoria inicial 2100 CIO
LD P_On
SET 2102.00  ; gate open
; rung 1
LD P_Off
SET 2102.01  ; Gate Close
; rung 2
LD T0215  ; Tiempo para hacer 0
OUT 2102.03  ; Reset counter 1
; rung 3
LD P_On
CALL Contador_1 : Conversion_Encoder (Encoder := 2122, Constante_conversion := +2,880000114, Encoder_en_mm => D2000)  ; Counter1 (módulo CT021), Encoder en milimetros
; rung 4: Habilitacion
LD Pulsador_abrir_sujetador  ; Llave de habilitación
OUT Hab_FILM  ; Habilitación proceso máquina film
; rung 5: Secuencia
LD P_On
MLPX(076) D100 #1000 W300  ; Pasos secuencia Maquina Film
; rung 6
LDNOT Hab_FILM  ; Habilitación proceso máquina film
BSET(071) &0 D100 D101  ; Pasos secuencia Maquina Film, Paso anterior
; rung 7: Paso 0 / Inicio secuencia
@LD Hab_FILM  ; Habilitación proceso máquina film
AND W300.00  ; Paso 0 maquina Film
MOV(021) &1 D100  ; Pasos secuencia Maquina Film
RSET 400.10  ; Cero carro OK

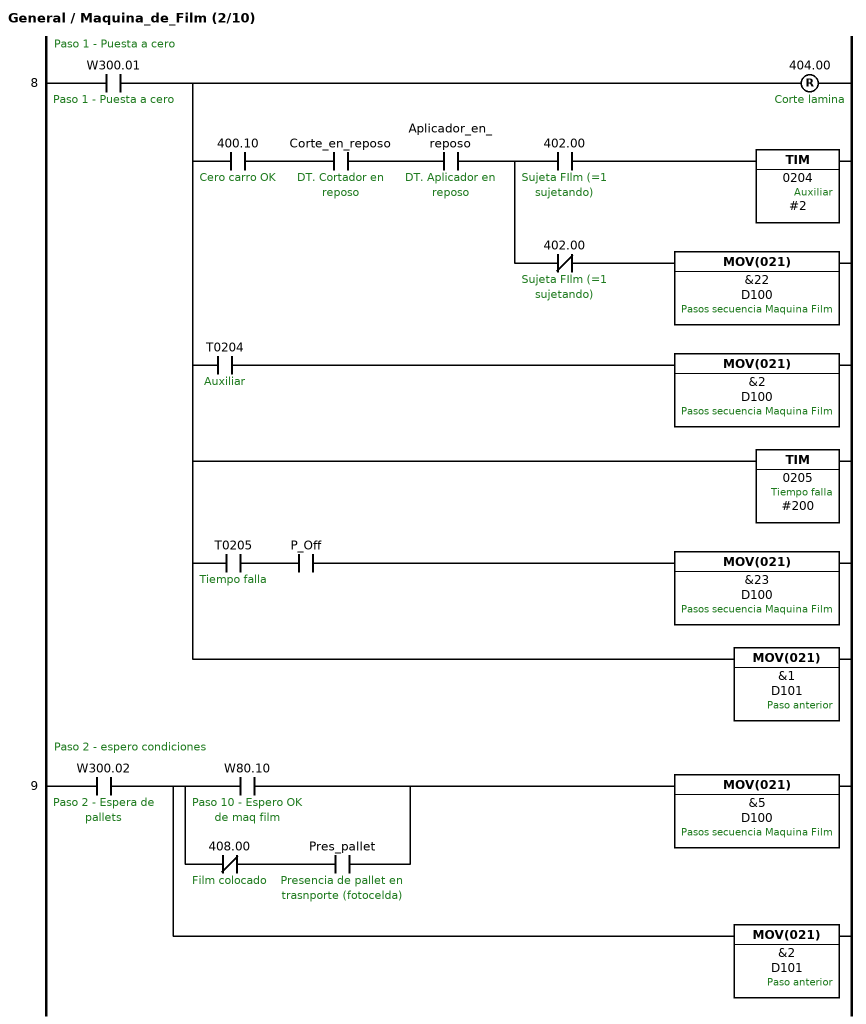
; rung 8: Paso 1 - Puesta a cero
LD W300.01  ; Paso 1 - Puesta a cero
OUT TR0
RSET 404.00  ; Corte lamina
AND 400.10  ; Cero carro OK
AND Corte_en_reposo  ; DT. Cortador en reposo
AND Aplicador_en_reposo  ; DT. Aplicador en reposo
OUT TR1
AND 402.00  ; Sujeta FIlm (=1 sujetando)
TIM 0204 #2  ; Auxiliar
LD TR1
ANDNOT 402.00  ; Sujeta FIlm (=1 sujetando)
MOV(021) &22 D100  ; Pasos secuencia Maquina Film
LD TR0
AND T0204  ; Auxiliar
MOV(021) &2 D100  ; Pasos secuencia Maquina Film
LD TR0
TIM 0205 #200  ; Tiempo falla
AND T0205  ; Tiempo falla
AND P_Off
MOV(021) &23 D100  ; Pasos secuencia Maquina Film
LD TR0
MOV(021) &1 D101  ; Paso anterior
; rung 9: Paso 2 - espero condiciones
LD W300.02  ; Paso 2 - Espera de pallets
OUT TR0
LD W80.10  ; Paso 10 - Espero OK de maq film
LDNOT 408.00  ; Film colocado
AND Pres_pallet  ; Presencia de pallet en trasnporte (fotocelda)
ORLD
ANDLD
MOV(021) &5 D100  ; Pasos secuencia Maquina Film
LD TR0
MOV(021) &2 D101  ; Paso anterior

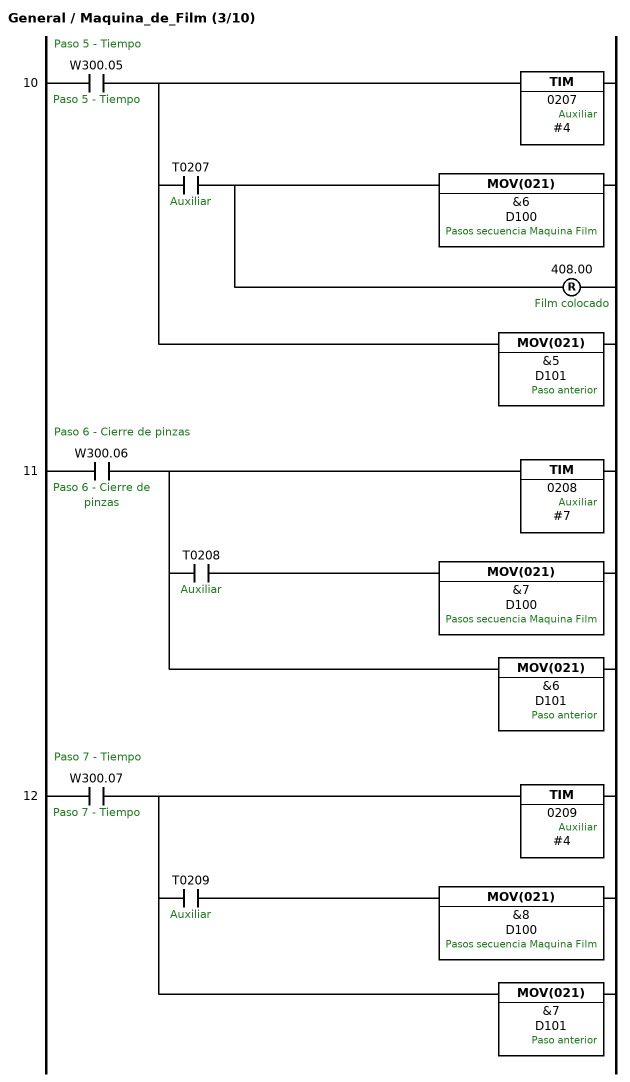
; rung 10: Paso 5 - Tiempo
LD W300.05  ; Paso 5 - Tiempo
OUT TR0
TIM 0207 #4  ; Auxiliar
AND T0207  ; Auxiliar
MOV(021) &6 D100  ; Pasos secuencia Maquina Film
RSET 408.00  ; Film colocado
LD TR0
MOV(021) &5 D101  ; Paso anterior
; rung 11: Paso 6 - Cierre de pinzas
LD W300.06  ; Paso 6 - Cierre de pinzas
OUT TR0
TIM 0208 #7  ; Auxiliar
AND T0208  ; Auxiliar
MOV(021) &7 D100  ; Pasos secuencia Maquina Film
LD TR0
MOV(021) &6 D101  ; Paso anterior
; rung 12: Paso 7 - Tiempo
LD W300.07  ; Paso 7 - Tiempo
OUT TR0
TIM 0209 #4  ; Auxiliar
AND T0209  ; Auxiliar
MOV(021) &8 D100  ; Pasos secuencia Maquina Film
LD TR0
MOV(021) &7 D101  ; Paso anterior

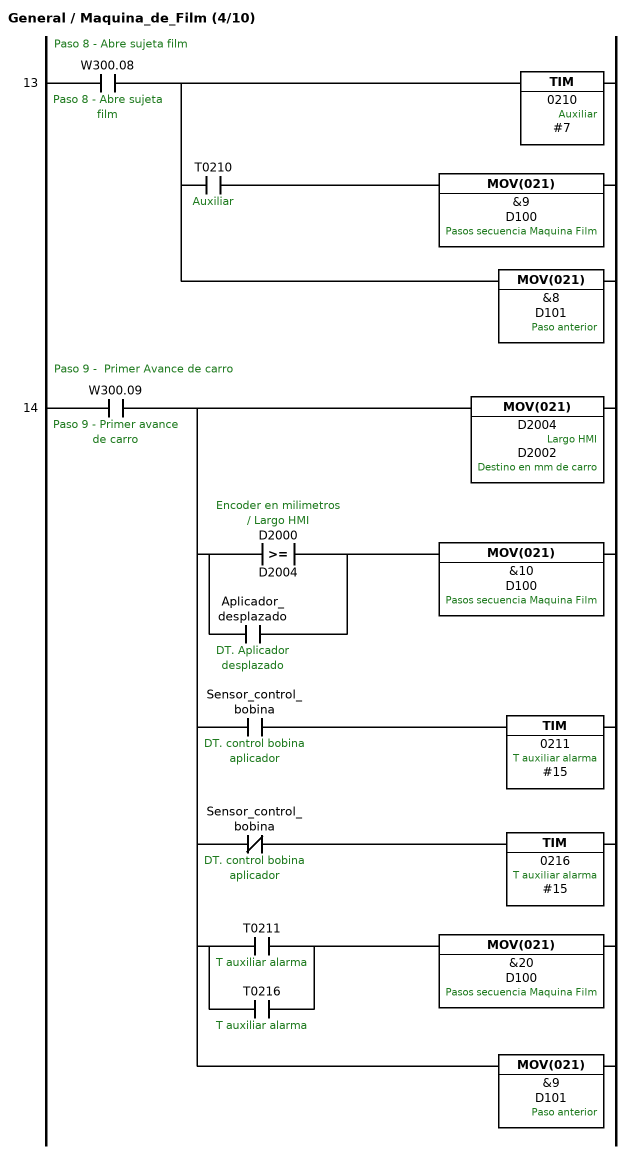
; rung 13: Paso 8 - Abre sujeta film
LD W300.08  ; Paso 8 - Abre sujeta film
OUT TR0
TIM 0210 #7  ; Auxiliar
AND T0210  ; Auxiliar
MOV(021) &9 D100  ; Pasos secuencia Maquina Film
LD TR0
MOV(021) &8 D101  ; Paso anterior
; rung 14: Paso 9 -  Primer Avance de carro
LD W300.09  ; Paso 9 - Primer avance de carro
OUT TR0
MOV(021) D2004 D2002  ; Largo HMI, Destino en mm de carro
LD>=SL(328) D2000 D2004  ; Encoder en milimetros, Largo HMI
OR Aplicador_desplazado  ; DT. Aplicador desplazado
ANDLD
MOV(021) &10 D100  ; Pasos secuencia Maquina Film
LD TR0
AND Sensor_control_bobina  ; DT. control bobina aplicador
TIM 0211 #15  ; T auxiliar alarma
LD TR0
ANDNOT Sensor_control_bobina  ; DT. control bobina aplicador
TIM 0216 #15  ; T auxiliar alarma
LD TR0
LD T0211  ; T auxiliar alarma
OR T0216  ; T auxiliar alarma
ANDLD
MOV(021) &20 D100  ; Pasos secuencia Maquina Film
LD TR0
MOV(021) &9 D101  ; Paso anterior

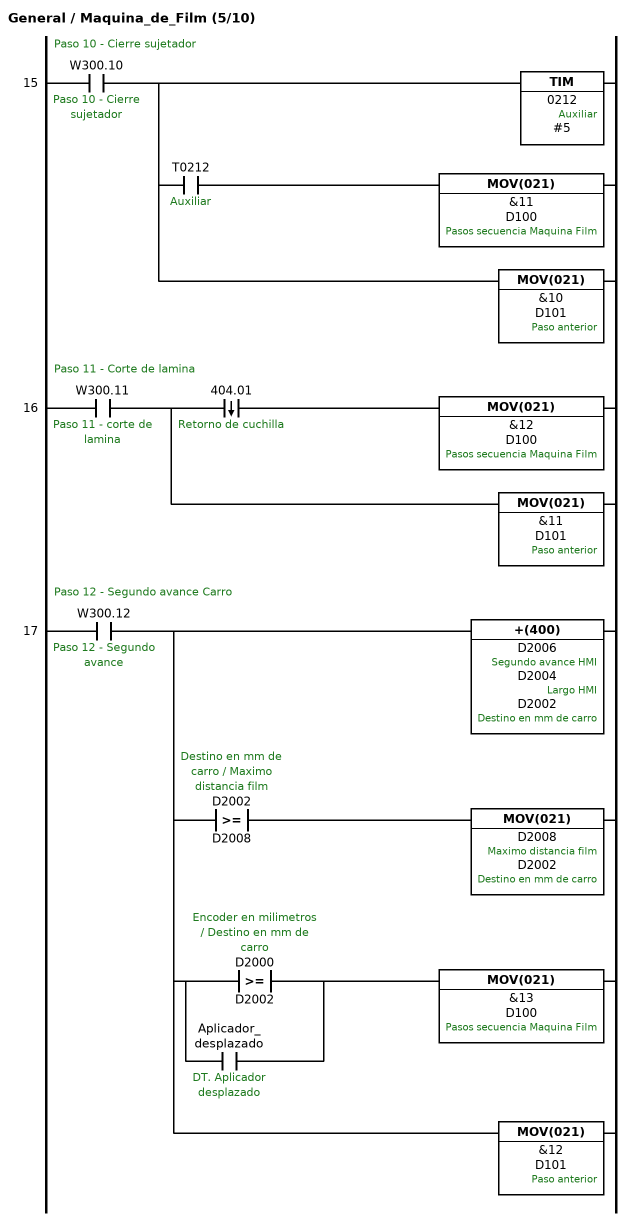
; rung 15: Paso 10 - Cierre sujetador
LD W300.10  ; Paso 10 - Cierre sujetador
OUT TR0
TIM 0212 #5  ; Auxiliar
AND T0212  ; Auxiliar
MOV(021) &11 D100  ; Pasos secuencia Maquina Film
LD TR0
MOV(021) &10 D101  ; Paso anterior
; rung 16: Paso 11 - Corte de lamina
LD W300.11  ; Paso 11 - corte de lamina
OUT TR0
%AND 404.01  ; Retorno de cuchilla
MOV(021) &12 D100  ; Pasos secuencia Maquina Film
LD TR0
MOV(021) &11 D101  ; Paso anterior
; rung 17: Paso 12 - Segundo avance Carro
LD W300.12  ; Paso 12 - Segundo avance
OUT TR0
+(400) D2006 D2004 D2002  ; Segundo avance HMI, Largo HMI, Destino en mm de carro
AND>=(325) D2002 D2008  ; Destino en mm de carro, Maximo distancia film
MOV(021) D2008 D2002  ; Maximo distancia film, Destino en mm de carro
LD TR0
LD>=(325) D2000 D2002  ; Encoder en milimetros, Destino en mm de carro
OR Aplicador_desplazado  ; DT. Aplicador desplazado
ANDLD
MOV(021) &13 D100  ; Pasos secuencia Maquina Film
LD TR0
MOV(021) &12 D101  ; Paso anterior

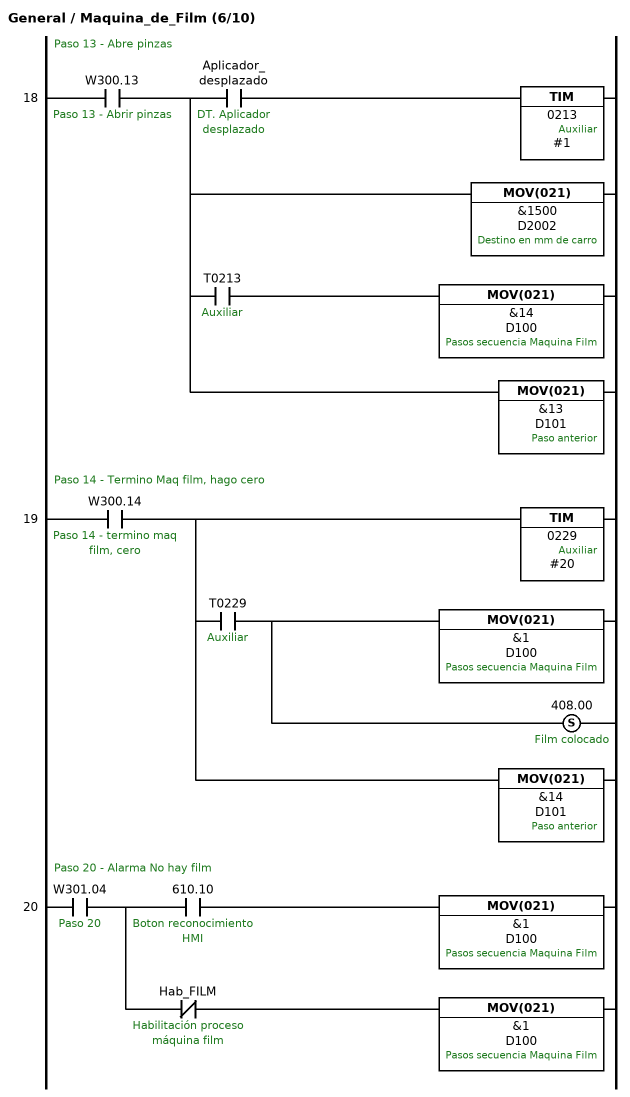
; rung 18: Paso 13 - Abre pinzas
LD W300.13  ; Paso 13 - Abrir pinzas
OUT TR0
AND Aplicador_desplazado  ; DT. Aplicador desplazado
TIM 0213 #1  ; Auxiliar
LD TR0
MOV(021) &1500 D2002  ; Destino en mm de carro
AND T0213  ; Auxiliar
MOV(021) &14 D100  ; Pasos secuencia Maquina Film
LD TR0
MOV(021) &13 D101  ; Paso anterior
; rung 19: Paso 14 - Termino Maq film, hago cero
LD W300.14  ; Paso 14 - termino maq film, cero
OUT TR0
TIM 0229 #20  ; Auxiliar
AND T0229  ; Auxiliar
MOV(021) &1 D100  ; Pasos secuencia Maquina Film
SET 408.00  ; Film colocado
LD TR0
MOV(021) &14 D101  ; Paso anterior
; rung 20: Paso 20 - Alarma No hay film
LD W301.04  ; Paso 20
OUT TR0
AND 610.10  ; Boton reconocimiento HMI
MOV(021) &1 D100  ; Pasos secuencia Maquina Film
LD TR0
ANDNOT Hab_FILM  ; Habilitación proceso máquina film
MOV(021) &1 D100  ; Pasos secuencia Maquina Film

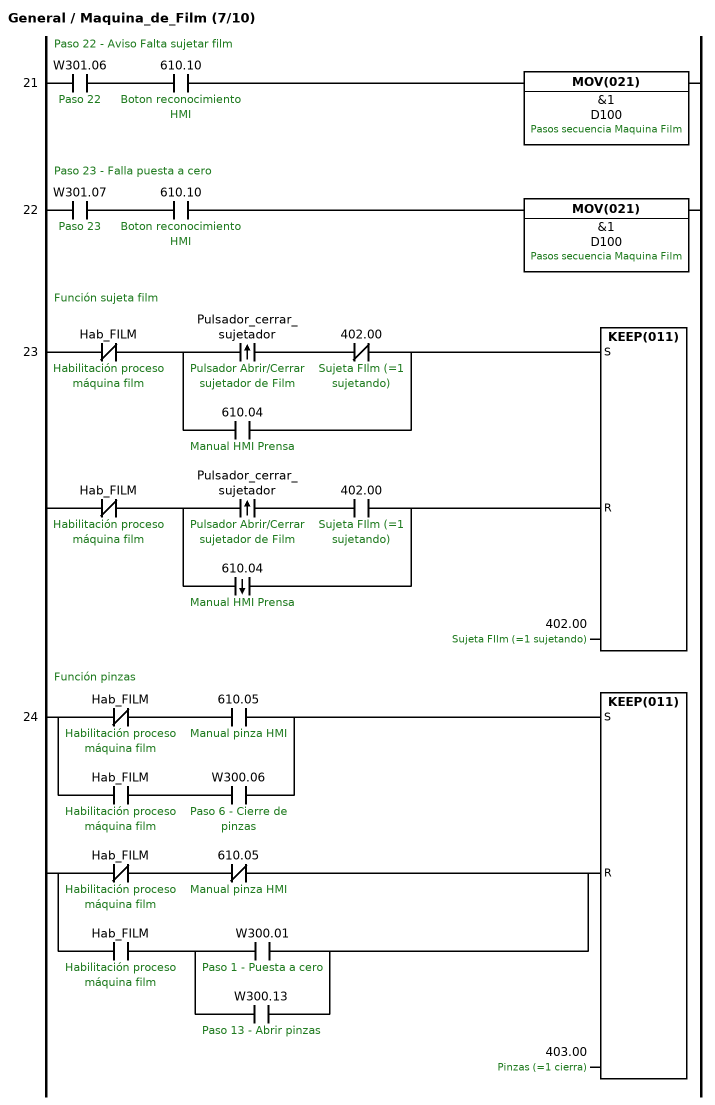
; rung 21: Paso 22 - Aviso Falta sujetar film
LD W301.06  ; Paso 22
AND 610.10  ; Boton reconocimiento HMI
MOV(021) &1 D100  ; Pasos secuencia Maquina Film
; rung 22: Paso 23 - Falla puesta a cero
LD W301.07  ; Paso 23
AND 610.10  ; Boton reconocimiento HMI
MOV(021) &1 D100  ; Pasos secuencia Maquina Film
; rung 23: Función sujeta film
LDNOT Hab_FILM  ; Habilitación proceso máquina film
@LD Pulsador_cerrar_sujetador  ; Pulsador Abrir/Cerrar sujetador de Film
ANDNOT 402.00  ; Sujeta FIlm (=1 sujetando)
OR 610.04  ; Manual HMI Prensa
ANDLD
LDNOT Hab_FILM  ; Habilitación proceso máquina film
@LD Pulsador_cerrar_sujetador  ; Pulsador Abrir/Cerrar sujetador de Film
AND 402.00  ; Sujeta FIlm (=1 sujetando)
%OR 610.04  ; Manual HMI Prensa
ANDLD
KEEP(011) 402.00  ; Sujeta FIlm (=1 sujetando)
; rung 24: Función pinzas
LDNOT Hab_FILM  ; Habilitación proceso máquina film
AND 610.05  ; Manual pinza HMI
LD Hab_FILM  ; Habilitación proceso máquina film
AND W300.06  ; Paso 6 - Cierre de pinzas
ORLD
LDNOT Hab_FILM  ; Habilitación proceso máquina film
ANDNOT 610.05  ; Manual pinza HMI
LD Hab_FILM  ; Habilitación proceso máquina film
LD W300.01  ; Paso 1 - Puesta a cero
OR W300.13  ; Paso 13 - Abrir pinzas
ANDLD
ORLD
KEEP(011) 403.00  ; Pinzas (=1 cierra)

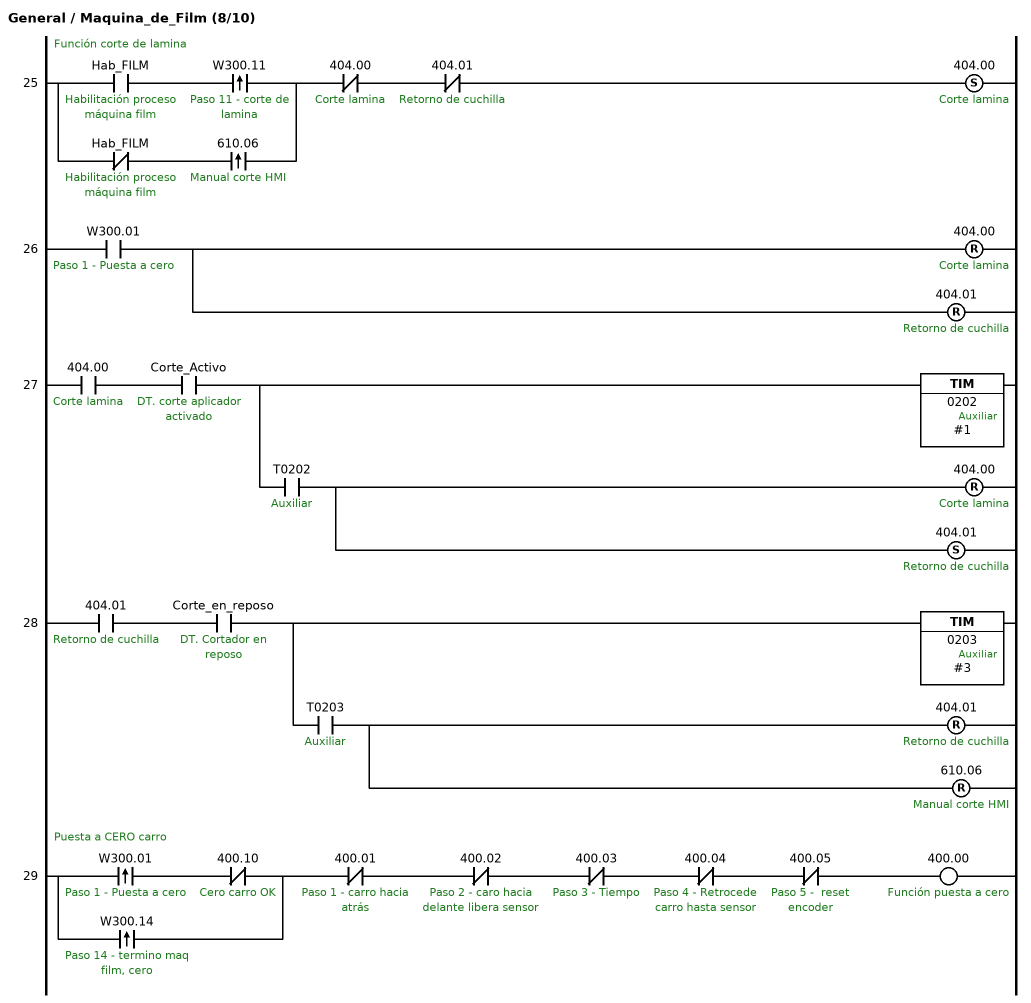
; rung 25: Función corte de lamina
LD Hab_FILM  ; Habilitación proceso máquina film
@AND W300.11  ; Paso 11 - corte de lamina
LDNOT Hab_FILM  ; Habilitación proceso máquina film
@AND 610.06  ; Manual corte HMI
ORLD
ANDNOT 404.00  ; Corte lamina
ANDNOT 404.01  ; Retorno de cuchilla
SET 404.00  ; Corte lamina
; rung 26
LD W300.01  ; Paso 1 - Puesta a cero
RSET 404.00  ; Corte lamina
RSET 404.01  ; Retorno de cuchilla
; rung 27
LD 404.00  ; Corte lamina
AND Corte_Activo  ; DT. corte aplicador activado
TIM 0202 #1  ; Auxiliar
AND T0202  ; Auxiliar
RSET 404.00  ; Corte lamina
SET 404.01  ; Retorno de cuchilla
; rung 28
LD 404.01  ; Retorno de cuchilla
AND Corte_en_reposo  ; DT. Cortador en reposo
TIM 0203 #3  ; Auxiliar
AND T0203  ; Auxiliar
RSET 404.01  ; Retorno de cuchilla
RSET 610.06  ; Manual corte HMI
; rung 29: Puesta a CERO carro
@LD W300.01  ; Paso 1 - Puesta a cero
ANDNOT 400.10  ; Cero carro OK
@OR W300.14  ; Paso 14 - termino maq film, cero
ANDNOT 400.01  ; Paso 1 - carro hacia atrás
ANDNOT 400.02  ; Paso 2 - caro hacia delante libera sensor
ANDNOT 400.03  ; Paso 3 - Tiempo
ANDNOT 400.04  ; Paso 4 - Retrocede carro hasta sensor
ANDNOT 400.05  ; Paso 5 -  reset encoder
OUT 400.00  ; Función puesta a cero

